	MW(WORD_STRONG := MesBlock1_Temp[1][  4], WORD_WEAK := MesBlock1_Temp[1][  3], VAR_OUT := MesDataExd.T1.MesI2);                       
	MW(WORD_STRONG := MesBlock1_Temp[1][  6], WORD_WEAK := MesBlock1_Temp[1][  5], VAR_OUT := MesDataExd.T1.MesI3);                       
	MW(WORD_STRONG := MesBlock1_Temp[1][  8], WORD_WEAK := MesBlock1_Temp[1][  7], VAR_OUT := MesDataExd.T1.MesU12);                      
	MW(WORD_STRONG := MesBlock1_Temp[1][ 10], WORD_WEAK := MesBlock1_Temp[1][  9], VAR_OUT := MesDataExd.T1.MesU23);                      
	MW(WORD_STRONG := MesBlock1_Temp[1][ 12], WORD_WEAK := MesBlock1_Temp[1][ 11], VAR_OUT := MesDataExd.T1.MesU31);                      
	MW(WORD_STRONG := MesBlock1_Temp[1][ 14], WORD_WEAK := MesBlock1_Temp[1][ 13], VAR_OUT := MesDataExd.T2.MesI1);                       
	MW(WORD_STRONG := MesBlock1_Temp[1][ 16], WORD_WEAK := MesBlock1_Temp[1][ 15], VAR_OUT := MesDataExd.T2.MesI2);                       
	MW(WORD_STRONG := MesBlock1_Temp[1][ 18], WORD_WEAK := MesBlock1_Temp[1][ 17], VAR_OUT := MesDataExd.T2.MesI3);                       
	MW(WORD_STRONG := MesBlock1_Temp[1][ 20], WORD_WEAK := MesBlock1_Temp[1][ 19], VAR_OUT := MesDataExd.T2.MesU12);                      
	MW(WORD_STRONG := MesBlock1_Temp[1][ 22], WORD_WEAK := MesBlock1_Temp[1][ 21], VAR_OUT := MesDataExd.T2.MesU23);                      
	MW(WORD_STRONG := MesBlock1_Temp[1][ 24], WORD_WEAK := MesBlock1_Temp[1][ 23], VAR_OUT := MesDataExd.T2.MesU31);                      
	MW(WORD_STRONG := MesBlock1_Temp[1][ 26], WORD_WEAK := MesBlock1_Temp[1][ 25], VAR_OUT := MesDataExd.T2.MesFreq );                             
	MW(WORD_STRONG := MesBlock1_Temp[1][ 28], WORD_WEAK := MesBlock1_Temp[1][ 27], VAR_OUT := MesDataExd.F11.MesEActProd);                                 
	MW(WORD_STRONG := MesBlock1_Temp[1][ 30], WORD_WEAK := MesBlock1_Temp[1][ 29], VAR_OUT := MesDataExd.F11.MesEActCons);                                 
	MW(WORD_STRONG := MesBlock1_Temp[1][ 32], WORD_WEAK := MesBlock1_Temp[1][ 31], VAR_OUT := MesDataExd.F11.MesEReactProd);               
	MW(WORD_STRONG := MesBlock1_Temp[1][ 34], WORD_WEAK := MesBlock1_Temp[1][ 33], VAR_OUT := MesDataExd.F11.MesEReactCons);                    
	MW(WORD_STRONG := MesBlock1_Temp[1][ 36], WORD_WEAK := MesBlock1_Temp[1][ 35], VAR_OUT := MesDataExd.F11.MesP);                       
	MW(WORD_STRONG := MesBlock1_Temp[1][ 38], WORD_WEAK := MesBlock1_Temp[1][ 37], VAR_OUT := MesDataExd.F11.MesQ);                       
	MW(WORD_STRONG := MesBlock1_Temp[1][ 40], WORD_WEAK := MesBlock1_Temp[1][ 39], VAR_OUT := MesDataExd.F11.MesU12);                     
	MW(WORD_STRONG := MesBlock1_Temp[1][ 42], WORD_WEAK := MesBlock1_Temp[1][ 41], VAR_OUT := MesDataExd.F11.MesU23);                     
	MW(WORD_STRONG := MesBlock1_Temp[1][ 44], WORD_WEAK := MesBlock1_Temp[1][ 43], VAR_OUT := MesDataExd.F11.MesU31);                     
	MW(WORD_STRONG := MesBlock1_Temp[1][ 46], WORD_WEAK := MesBlock1_Temp[1][ 45], VAR_OUT := MesDataExd.F11.MesV1);                      
	MW(WORD_STRONG := MesBlock1_Temp[1][ 48], WORD_WEAK := MesBlock1_Temp[1][ 47], VAR_OUT := MesDataExd.F11.MesV2);                      
	MW(WORD_STRONG := MesBlock1_Temp[1][ 50], WORD_WEAK := MesBlock1_Temp[1][ 49], VAR_OUT := MesDataExd.F11.MesV3);                      
	MW(WORD_STRONG := MesBlock1_Temp[1][ 52], WORD_WEAK := MesBlock1_Temp[1][ 51], VAR_OUT := MesDataExd.F11.MesI1);                      
	MW(WORD_STRONG := MesBlock1_Temp[1][ 54], WORD_WEAK := MesBlock1_Temp[1][ 53], VAR_OUT := MesDataExd.F11.MesI2);                      
	MW(WORD_STRONG := MesBlock1_Temp[1][ 56], WORD_WEAK := MesBlock1_Temp[1][ 55], VAR_OUT := MesDataExd.F11.MesI3);                   
	MW(WORD_STRONG := MesBlock1_Temp[1][ 58], WORD_WEAK := MesBlock1_Temp[1][ 57], VAR_OUT := MesDataExd.F11.MesFreq);                    
	MW(WORD_STRONG := MesBlock1_Temp[1][ 60], WORD_WEAK := MesBlock1_Temp[1][ 59], VAR_OUT := MesDataExd.F11.MesCosPhi);                
	MW(WORD_STRONG := MesBlock1_Temp[1][ 62], WORD_WEAK := MesBlock1_Temp[1][ 61], VAR_OUT := MesDataExd.F15.MesP);                 
	MW(WORD_STRONG := MesBlock1_Temp[1][ 64], WORD_WEAK := MesBlock1_Temp[1][ 63], VAR_OUT := MesDataExd.F15.MesQ);                 
	MW(WORD_STRONG := MesBlock1_Temp[1][ 66], WORD_WEAK := MesBlock1_Temp[1][ 65],  VAR_OUT :=MesDataExd.F15.MesI1);                     
	MW(WORD_STRONG := MesBlock1_Temp[1][ 68], WORD_WEAK := MesBlock1_Temp[1][ 67],  VAR_OUT :=MesDataExd.F15.MesI2);                  
	MW(WORD_STRONG := MesBlock1_Temp[1][ 70], WORD_WEAK := MesBlock1_Temp[1][ 69],  VAR_OUT :=MesDataExd.F15.MesI3);                  
	MW(WORD_STRONG := MesBlock1_Temp[1][ 72], WORD_WEAK := MesBlock1_Temp[1][ 71],  VAR_OUT :=MesDataExd.F15.MesU12);                 
	MW(WORD_STRONG := MesBlock1_Temp[1][ 74], WORD_WEAK := MesBlock1_Temp[1][ 73],  VAR_OUT :=MesDataExd.F15.MesU23);          
	MW(WORD_STRONG := MesBlock1_Temp[1][ 76], WORD_WEAK := MesBlock1_Temp[1][ 75],  VAR_OUT :=MesDataExd.F15.MesU31);    
	MW(WORD_STRONG := MesBlock1_Temp[1][ 78], WORD_WEAK := MesBlock1_Temp[1][ 77],  VAR_OUT :=MesDataExd.F15.MesV1);       
	MW(WORD_STRONG := MesBlock1_Temp[1][ 78], WORD_WEAK := MesBlock1_Temp[1][ 79],  VAR_OUT :=MesDataExd.F15.MesV2);       
	MW(WORD_STRONG := MesBlock1_Temp[1][ 80], WORD_WEAK := MesBlock1_Temp[1][ 81],  VAR_OUT :=MesDataExd.F15.MesV3);                
	MW(WORD_STRONG := MesBlock1_Temp[1][ 84], WORD_WEAK := MesBlock1_Temp[1][ 85],  VAR_OUT :=MesDataExd.F15.MesFreq);   

                    
	MW(WORD_STRONG := MesBlock1_Temp[2][ 22], WORD_WEAK := MesBlock1_Temp[2][21], VAR_OUT := MesDataExd.F21.MesEActProd);                      
	MW(WORD_STRONG := MesBlock1_Temp[2][ 24], WORD_WEAK := MesBlock1_Temp[2][23], VAR_OUT := MesDataExd.F21.MesEActCons);                      
	MW(WORD_STRONG := MesBlock1_Temp[2][ 26], WORD_WEAK := MesBlock1_Temp[2][25], VAR_OUT := MesDataExd.F21.MesEReactProd);                    
	MW(WORD_STRONG := MesBlock1_Temp[2][ 28], WORD_WEAK := MesBlock1_Temp[2][27], VAR_OUT := MesDataExd.F21.MesEReactCons);                    
	MW(WORD_STRONG := MesBlock1_Temp[2][ 30], WORD_WEAK := MesBlock1_Temp[2][29], VAR_OUT := MesDataExd.F21.MesP);                            
	MW(WORD_STRONG := MesBlock1_Temp[2][ 32], WORD_WEAK := MesBlock1_Temp[2][31], VAR_OUT := MesDataExd.F21.MesQ);                            
	MW(WORD_STRONG := MesBlock1_Temp[2][ 34], WORD_WEAK := MesBlock1_Temp[2][33], VAR_OUT := MesDataExd.F21.MesU12);                          
	MW(WORD_STRONG := MesBlock1_Temp[2][ 36], WORD_WEAK := MesBlock1_Temp[2][35], VAR_OUT := MesDataExd.F21.MesU23);                          
	MW(WORD_STRONG := MesBlock1_Temp[2][ 38], WORD_WEAK := MesBlock1_Temp[2][37], VAR_OUT := MesDataExd.F21.MesU31);                          
	MW(WORD_STRONG := MesBlock1_Temp[2][ 40], WORD_WEAK := MesBlock1_Temp[2][39], VAR_OUT := MesDataExd.F21.MesV1);                           
	MW(WORD_STRONG := MesBlock1_Temp[2][ 42], WORD_WEAK := MesBlock1_Temp[2][41], VAR_OUT := MesDataExd.F21.MesV2);                           
	MW(WORD_STRONG := MesBlock1_Temp[2][ 44], WORD_WEAK := MesBlock1_Temp[2][43], VAR_OUT := MesDataExd.F21.MesV3);                           
	MW(WORD_STRONG := MesBlock1_Temp[2][ 46], WORD_WEAK := MesBlock1_Temp[2][45], VAR_OUT := MesDataExd.F21.MesI1);                           
	MW(WORD_STRONG := MesBlock1_Temp[2][ 48], WORD_WEAK := MesBlock1_Temp[2][47], VAR_OUT := MesDataExd.F21.MesI2);                           
	MW(WORD_STRONG := MesBlock1_Temp[2][ 50], WORD_WEAK := MesBlock1_Temp[2][49], VAR_OUT := MesDataExd.F21.MesI3);                           
	MW(WORD_STRONG := MesBlock1_Temp[2][ 52], WORD_WEAK := MesBlock1_Temp[2][51], VAR_OUT := MesDataExd.F21.MesFreq);                         
	MW(WORD_STRONG := MesBlock1_Temp[2][ 54], WORD_WEAK := MesBlock1_Temp[2][53], VAR_OUT := MesDataExd.F21.MesCosPhi);                       
	MW(WORD_STRONG := MesBlock1_Temp[2][ 56], WORD_WEAK := MesBlock1_Temp[2][55], VAR_OUT := MesDataExd.F22.MesEActProd);                      
	MW(WORD_STRONG := MesBlock1_Temp[2][ 58], WORD_WEAK := MesBlock1_Temp[2][57], VAR_OUT := MesDataExd.F22.MesEActCons);                      
	MW(WORD_STRONG := MesBlock1_Temp[2][ 60], WORD_WEAK := MesBlock1_Temp[2][59], VAR_OUT := MesDataExd.F22.MesEReactProd);                    
	MW(WORD_STRONG := MesBlock1_Temp[2][ 62], WORD_WEAK := MesBlock1_Temp[2][61], VAR_OUT := MesDataExd.F22.MesEReactCons);                    
	MW(WORD_STRONG := MesBlock1_Temp[2][ 64], WORD_WEAK := MesBlock1_Temp[2][63], VAR_OUT := MesDataExd.F22.MesP);                            
	MW(WORD_STRONG := MesBlock1_Temp[2][ 66], WORD_WEAK := MesBlock1_Temp[2][65], VAR_OUT := MesDataExd.F22.MesQ);                            
	MW(WORD_STRONG := MesBlock1_Temp[2][ 68], WORD_WEAK := MesBlock1_Temp[2][67], VAR_OUT := MesDataExd.F22.MesU12);                          
	MW(WORD_STRONG := MesBlock1_Temp[2][ 70], WORD_WEAK := MesBlock1_Temp[2][69], VAR_OUT := MesDataExd.F22.MesU23);                          
	MW(WORD_STRONG := MesBlock1_Temp[2][ 72], WORD_WEAK := MesBlock1_Temp[2][71], VAR_OUT := MesDataExd.F22.MesU31);                          
	MW(WORD_STRONG := MesBlock1_Temp[2][ 74], WORD_WEAK := MesBlock1_Temp[2][73], VAR_OUT := MesDataExd.F22.MesV1);                           
	MW(WORD_STRONG := MesBlock1_Temp[2][ 76], WORD_WEAK := MesBlock1_Temp[2][75], VAR_OUT := MesDataExd.F22.MesV2);                           
	MW(WORD_STRONG := MesBlock1_Temp[2][ 78], WORD_WEAK := MesBlock1_Temp[2][77], VAR_OUT := MesDataExd.F22.MesV3);                           
	MW(WORD_STRONG := MesBlock1_Temp[2][ 80], WORD_WEAK := MesBlock1_Temp[2][79], VAR_OUT := MesDataExd.F22.MesI1);                           
	MW(WORD_STRONG := MesBlock1_Temp[2][ 82], WORD_WEAK := MesBlock1_Temp[2][81], VAR_OUT := MesDataExd.F22.MesI2);                           
	MW(WORD_STRONG := MesBlock1_Temp[2][ 84], WORD_WEAK := MesBlock1_Temp[2][83], VAR_OUT := MesDataExd.F22.MesI3);                           
	MW(WORD_STRONG := MesBlock1_Temp[2][ 86], WORD_WEAK := MesBlock1_Temp[2][85], VAR_OUT := MesDataExd.F22.MesFreq);                         
	MW(WORD_STRONG := MesBlock1_Temp[2][ 88], WORD_WEAK := MesBlock1_Temp[2][87], VAR_OUT := MesDataExd.F22.MesCosPhi); 

	MW(WORD_WEAK := MesBlock1_Temp[3][ 1], WORD_STRONG := MesBlock1_Temp[3][ 2], VAR_OUT := MesDataExd.T4.MesU12);
	MW(WORD_WEAK := MesBlock1_Temp[3][ 3], WORD_STRONG := MesBlock1_Temp[3][ 4], VAR_OUT := MesDataExd.T4.MesU23);
	MW(WORD_WEAK := MesBlock1_Temp[3][ 5], WORD_STRONG := MesBlock1_Temp[3][ 6], VAR_OUT := MesDataExd.T4.MesU31);
	                                                                              
	MW(WORD_WEAK := MesBlock1_Temp[4][ 1], WORD_STRONG := MesBlock1_Temp[4][ 2], VAR_OUT := MesDataExd.T5.MesU12);
	MW(WORD_WEAK := MesBlock1_Temp[4][ 3], WORD_STRONG := MesBlock1_Temp[4][ 4], VAR_OUT := MesDataExd.T5.MesU23);
	MW(WORD_WEAK := MesBlock1_Temp[4][ 5], WORD_STRONG := MesBlock1_Temp[4][ 6], VAR_OUT := MesDataExd.T5.MesU31);
	
MesDataExd.F11.MesU := (MesDataExd.F11.MesU12 + MesDataExd.F11.MesU23 + MesDataExd.F11.MesU31)/3 ;
MesDataExd.F11.MesI := (MesDataExd.F11.MesI1 + MesDataExd.F11.MesI2 + MesDataExd.F11.MesI3)/3 ;
MesDataExd.F11.MesV := (MesDataExd.F11.MesV1 + MesDataExd.F11.MesV2 + MesDataExd.F11.MesV3)/3 ;

MesDataExd.F15.MesU := (MesDataExd.F15.MesU12 + MesDataExd.F15.MesU23 + MesDataExd.F15.MesU31)/3 ;
MesDataExd.F15.MesI := (MesDataExd.F15.MesI1 + 	MesDataExd.F15.MesI2 + 	MesDataExd.F15.MesI3)/3 ;
MesDataExd.F15.MesV := (MesDataExd.F15.MesV1 + 	MesDataExd.F15.MesV2 + 	MesDataExd.F15.MesV3)/3 ;

MesDataExd.F21.MesU := (MesDataExd.F21.MesU12 + MesDataExd.F21.MesU23 + MesDataExd.F21.MesU31)/3 ;
MesDataExd.F21.MesI := (MesDataExd.F21.MesI1 + 	MesDataExd.F21.MesI2 + 	MesDataExd.F21.MesI3)/3 ;
MesDataExd.F21.MesV := (MesDataExd.F21.MesV1 + 	MesDataExd.F21.MesV2 + 	MesDataExd.F21.MesV3)/3 ;

MesDataExd.F22.MesU := (MesDataExd.F22.MesU12 + MesDataExd.F22.MesU23 + MesDataExd.F22.MesU31)/3 ;
MesDataExd.F22.MesI := (MesDataExd.F22.MesI1 + 	MesDataExd.F22.MesI2 + 	MesDataExd.F22.MesI3)/3 ;
MesDataExd.F22.MesV := (MesDataExd.F22.MesV1 + 	MesDataExd.F22.MesV2 + 	MesDataExd.F22.MesV3)/3 ;

MesDataExd.T1.MesU := (MesDataExd.T1.MesU12 + 	MesDataExd.T1.MesU23 + 	MesDataExd.T1.MesU31)/3 ;
MesDataExd.T1.MesI := (MesDataExd.T1.MesI1 + 	MesDataExd.T1.MesI2 + 	MesDataExd.T1.MesI3)/3 ;
MesDataExd.T1.MesV := (MesDataExd.T1.MesV1 + 	MesDataExd.T1.MesV2 + 	MesDataExd.T1.MesV3)/3 ;

MesDataExd.T2.MesU := (MesDataExd.T2.MesU12 + 	MesDataExd.T2.MesU23 + 	MesDataExd.T2.MesU31)/3 ;
MesDataExd.T2.MesI := (MesDataExd.T2.MesI1 + 	MesDataExd.T2.MesI2 + 	MesDataExd.T2.MesI3)/3 ;
MesDataExd.T2.MesV := (MesDataExd.T2.MesV1 + 	MesDataExd.T2.MesV2 + 	MesDataExd.T2.MesV3)/3 ;

MesDataExd.T4.MesU := (MesDataExd.T4.MesU12 + 	MesDataExd.T4.MesU23 + 	MesDataExd.T4.MesU31)/3 ;
MesDataExd.T5.MesU := (MesDataExd.T5.MesU12 + 	MesDataExd.T5.MesU23 + 	MesDataExd.T5.MesU31)/3 ;
END_METHOD

END_FUNCTION_BLOCK

// ---- 01_Equipement_Library/Operation Meter/FB_PM_520x230.TcPOU
FUNCTION_BLOCK FB_PM_520x230 EXTENDS FB_PM_Base
//////////////////
// Measurement Solution based on Digiware, but access through PMS Socomec
//////////////////
VAR CONSTANT
	// Characteristics of the object (Same for all instances)
			
END_VAR

VAR_INPUT PERSISTENT
	// Parameters of the Object (instance specific) 
	{attribute 'OPC.UA.DA' := '1'} 
	ParamUnitID					: BYTE := 1 ;									// (NA)unit ID
	ParamInInterfaceSub			: BOOL := TRUE; 								// Serial interface RS422/RS485 TYPE (0:EL6021,1:SUB9)			
END_VAR

VAR_OUTPUT
	//Child objects
	
END_VAR


VAR_INPUT 
			MesDataExd				: PM_Standard;								// (NA) Structure of the PM3250
END_VAR

VAR
	//M_ALARMMANAGEMENT VARIABLES//
	                                                    								
                                                        								

	//M_READ VARIABLES//
		ModbusRTU					: FB_ModbusRTU;								// (NA) FB for Modbus Reading


		ObjectCom					: INT;										// (NA) Sequence index
									
		Busy						: BOOL;
		StepRead					: UINT;										// (NA) Step for reading 2 blocks of registers
		AX_TrigRead					: ARRAY[1..1] OF R_trig;
		MbStruct					: ARRAY[1..1] OF Struct_InputRTU;	
		MesBlock					: ARRAY[1..1] OF ARRAY[1..120] OF WORD;	
		AX_Addr						: ARRAY[1..1] OF UINT 	:= [19000];
		AX_Qty						: ARRAY[1..1] OF UINT	:= [86];
		AX_UnitId					: ARRAY[1..1] OF BYTE	:= [1];
		AX_Function					: ARRAY[1..1] OF UINT	:= [4];	
		AX_Priority					: ARRAY[1..1] OF UINT	:= [1];
		KK							: INT;
		ComError 					: BOOL;
	//M_INIT VARIABLES //
		OutFBCompleteted			: BOOL;
	// M_EXECUTE VARIABLES //
		
                              

 
END_VAR

METHOD M_AlarmManagement
//////////////////
// Digiware measurement tool alarm and warning management
/////////////////

VAR 
	// Method local variables (reinitialized at each cycle) 
	FB_AlarmCodeManager			: FB_AlarmCodeManager ; 
	
	KK							: BYTE ;		// For loop
	
	CMWarning					: BOOL;			// At least one Digiware device in Alarm
	CMAlarm						: BOOL;			// At least one Digiware device in Alarm
	
END_VAR
//ComError 	:= MbStruct[1].OutError^;
	
TON_ComAlarm(IN:= ComError , PT:= ParamTempoComAlarm, Q=>MesDataExd.MesData.MesAlarmCom) ;	
TON_ComWarning(IN:= ComError  , PT:= ParamTempoComAlarm, Q=>MesWarningCom) ;	

//					General com alarm : All the read FB fucked up


// ALARM CODE //
	FB_AlarmCodeManager(
		bAlarm1			:= MesDataExd.MesData.MesAlarmCom  , 					// Communication Alarm #COM
		bAlarm2			:=FALSE, 		// 
		bAlarm3			:=FALSE, 		// 
		bAlarm4			:=FALSE, 		// 
		bAlarm5			:=FALSE, //
		bAlarm6			:=FALSE, //
		bAlarm7			:=FALSE, //
		bAlarm8			:=FALSE, //
		bAlarm9			:=FALSE, //
		bAlarm10		:=FALSE, //
		bAlarm11		:=FALSE, //
		bAlarm12		:=FALSE, //
		bAlarm13		:=FALSE, //
		bAlarm14		:=FALSE, //
		bAlarm15		:= FALSE , 			// 			 
		wAlarmCode		=>MesDataExd.MesData.MesAlarmCode);

// WARNING CODE //
	FB_AlarmCodeManager(		
		bAlarm1			:=MesWarningCom	,				 // Communication Warning #COM
		bAlarm2			:=FALSE, 		// 
		bAlarm3			:=FALSE, 		// 
		bAlarm4			:=FALSE, 		// 
		bAlarm5			:=FALSE, //
		bAlarm6			:=FALSE, //
		bAlarm7			:=FALSE, //
		bAlarm8			:=FALSE, //
		bAlarm9			:=FALSE, //
		bAlarm10		:=FALSE, //
		bAlarm11		:=FALSE, //
		bAlarm12		:=FALSE, //
		bAlarm13		:=FALSE, //
		bAlarm14		:=FALSE, //
		bAlarm15		:=FALSE, //
		wAlarmCode		=>MesDataExd.MesData.MesWarningCode);		

// EVENT CODE //
END_METHOD

METHOD M_CP
//////////////////
//  Emulator
/////////////////

VAR 
	// Method local variables (reinitialized at each cycle) 
	
END_VAR


SUPER^.M_CP() ; 




Trig_Cmd_Read(CLK:=IN_CmdToggleRead);
Trig_Cmd_Write(CLK:=IN_CmdToggleWrite);
	
IF Trig_Cmd_Read.Q THEN
	IN_CmdToggleRead := FALSE;
	MesDataExd.MesData.MesCP_Read := NOT MesDataExd.MesData.MesCP_Read;
END_IF


IF Trig_Cmd_Write.Q THEN
	IN_CmdToggleWrite := FALSE;
	MesDataExd.MesData.MesCP_Write := NOT MesDataExd.MesData.MesCP_Write;
END_IF
END_METHOD

METHOD M_Evaluate : BOOL
VAR_INPUT
END_VAR
END_METHOD

METHOD M_Execute
//////////////////
//  Method Calls 
/////////////////
VAR 
	// Method local variables (reinitialized at each cycle) 
	// EMULATOR
		Psoltot		: REAL;		// Total Solar Power . 
		KK			: BYTE;		// For Loop
	
END_VAR
// READING AND WRITING CLOCK //
	TP1(IN:=NOT TP1.Q , PT:= ParamClockReadTime);
	ClockRead 		:= TP1.Q;

// PERMANENT CONDITIONS //
	MesCP_Read 					:= TRUE  ; 
	
// METHODS CALLS //
	IF bInit THEN
		M_Init() ; 
		bInit					:= FALSE ; 
		
	END_IF

	M_Read() ; 
	
// EMULATOR COM READ  /////////////
	
	
	////////////////////
	M_AlarmManagement();
END_METHOD

METHOD M_Init
VAR 

END_VAR
//Modbus RTU Relay
FOR KK := 1 TO 1 DO 
	MbStruct[KK].InBuffer 		:= ADR(MesBlock[KK]);
	MbStruct[KK].InFunction 	:= AX_Function[KK];
	MbStruct[KK].InQuantity 	:= AX_Qty[KK];
	MbStruct[KK].InStartAddr 	:= AX_Addr[KK];
	MbStruct[KK].InUnitID 		:= AX_UnitId[KK];
	
END_FOR
END_METHOD

METHOD M_Read
//////////////////
//  Read Modbus Variable for PCS . 
/////////////////
VAR 
	// Method local variables (reinitialized at each cycle) 
	MW 					: FB_MergeWordsToFloat; 
	KK					: BYTE;  						// FOR Loop 

	
END_VAR
// CP-Read / Write 

MesDataExd.MesData.MesCP_Read := MesDataExd.MesData.MesCP_Read ; 
 

IF MesDataExd.MesData.MesCP_Read  THEN	

	ModbusRTU();
	
	
	FOR KK := 1 TO 1 DO
		AX_TrigRead[KK](CLK  :=ClockRead) ; // CalLocalTimeStruct.wSecond MOD 5 = 0);
		IF AX_TrigRead[KK].Q THEN
			ModbusRTU.M_AddAction_FIFO(InStruct := MbStruct[KK], InPriority := AX_Priority[KK]);
		END_IF
		MbStruct[KK].OutError			:= ADR(ComError);
	END_FOR  
							
	// PROPERTIES UPDATE // 
		// Block 1
	//MW( WORD_STRONG:= MesBlock_Temp[1][1], 	WORD_WEAK := MesBlock_Temp[1][2],	SIGNED:=TRUE, FIX:=0 , SIZE:=2, VAR_OUT := MesDataExd.MesData.MesI2);
		
	MW( WORD_STRONG:= MesBlock[1][1], 	WORD_WEAK := MesBlock[1][2], 	VAR_OUT:= MesDataExd.MesData.MesV1);
	MW( WORD_STRONG:= MesBlock[1][3], 	WORD_WEAK := MesBlock[1][4], 	VAR_OUT:= MesDataExd.MesData.MesV2);
	MW( WORD_STRONG:= MesBlock[1][5], 	WORD_WEAK := MesBlock[1][6], 	VAR_OUT:= MesDataExd.MesData.MesV3);
	MW( WORD_STRONG:= MesBlock[1][7], 	WORD_WEAK := MesBlock[1][8], 	VAR_OUT:= MesDataExd.MesData.MesU12);
	MW( WORD_STRONG:= MesBlock[1][9], 	WORD_WEAK := MesBlock[1][10], VAR_OUT:= MesDataExd.MesData.MesU23);
																					
	MW( WORD_STRONG:= MesBlock[1][11], 	WORD_WEAK := MesBlock[1][12], VAR_OUT:= MesDataExd.MesData.MesU31);
	MW( WORD_STRONG:= MesBlock[1][13], 	WORD_WEAK := MesBlock[1][14], VAR_OUT:= MesDataExd.MesData.MesI1);
	MW( WORD_STRONG:= MesBlock[1][15], 	WORD_WEAK := MesBlock[1][16], VAR_OUT:= MesDataExd.MesData.MesI2);
	MW( WORD_STRONG:= MesBlock[1][17], 	WORD_WEAK := MesBlock[1][18], VAR_OUT:= MesDataExd.MesData.MesI3);
	MW( WORD_STRONG:= MesBlock[1][19], 	WORD_WEAK := MesBlock[1][20], VAR_OUT:= MesDataExd.MesData.MesIN);
	MW( WORD_STRONG:= MesBlock[1][21], 	WORD_WEAK := MesBlock[1][22], VAR_OUT:= MesDataExd.MesData.MesP1);
	MW( WORD_STRONG:= MesBlock[1][23], 	WORD_WEAK := MesBlock[1][24], VAR_OUT:= MesDataExd.MesData.MesP2);
	MW( WORD_STRONG:= MesBlock[1][25], 	WORD_WEAK := MesBlock[1][26], VAR_OUT:= MesDataExd.MesData.MesP3);
																					
	MW( WORD_STRONG:= MesBlock[1][27], 	WORD_WEAK := MesBlock[1][28], VAR_OUT:= MesDataExd.MesData.MesP);
	MW( WORD_STRONG:= MesBlock[1][35], 	WORD_WEAK := MesBlock[1][36], VAR_OUT:= MesDataExd.MesData.MesS);
	MW( WORD_STRONG:= MesBlock[1][43], 	WORD_WEAK := MesBlock[1][44], VAR_OUT:= MesDataExd.MesData.MesQ);
	
	//MW( WORD_STRONG_F:= MesBlock[1][7], 	WORD_WEAK_F := MesBlock[1][8], NUMBER_F= MesDataExd.MesData.MesP);
	//MW( WORD_STRONG_F:= MesBlock[1][9], 	WORD_WEAK_F := MesBlock[1][10], NUMBER_F= MesDataExd.MesData.MesQ1);
	//MW( WORD_STRONG_F:= MesBlock[1][11], 	WORD_WEAK_F := MesBlock[1][12], NUMBER_F= MesDataExd.MesData.MesQ2);
	//MW( WORD_STRONG_F:= MesBlock[1][13], 	WORD_WEAK_F := MesBlock[1][14], NUMBER_F= MesDataExd.MesData.MesQ3);
	//MW( WORD_STRONG_F:= MesBlock[1][15], 	WORD_WEAK_F := MesBlock[1][16], NUMBER_F= MesDataExd.MesData.MesQ);
	//MW( WORD_STRONG_F:= MesBlock[1][23], 	WORD_WEAK_F := MesBlock[1][24], NUMBER_F= MesDataExd.MesData.MesS);
	
	//MW( WORD_STRONG_F:= MesBlock_Temp[4][1], 	WORD_WEAK_F := MesBlock_Temp[4][2], NUMBER_F= MesDataExd.MesData.MesTanPhi);
	//MW( WORD_STRONG_F:= MesBlock_Temp[4][3], 	WORD_WEAK_F := MesBlock_Temp[4][4], NUMBER_F= MesDataExd.MesData.MesFreq);
	//
	//MW( WORD_STRONG_F:= MesBlock_Temp[3][1], 	WORD_WEAK_F := MesBlock_Temp[3][2], NUMBER_F= MesDataExd.MesData.MesEActProd);
	//MW( WORD_STRONG_F:= MesBlock_Temp[3][3], 	WORD_WEAK_F := MesBlock_Temp[3][4], NUMBER_F= MesDataExd.MesData.MesEActCons);
	//MW( WORD_STRONG_F:= MesBlock_Temp[3][5], 	WORD_WEAK_F := MesBlock_Temp[3][6], NUMBER_F= MesDataExd.MesData.MesEReactProd);
	//MW( WORD_STRONG_F:= MesBlock_Temp[3][7], 	WORD_WEAK_F := MesBlock_Temp[3][8], NUMBER_F= MesDataExd.MesData.MesEReactCons);
	//MW( WORD_STRONG:= MesBlock_Temp[4][3], 	WORD_WEAK := MesBlock_Temp[4][4],	SIGNED:=TRUE, FIX:=0 , SIZE:=2, VAR_OUT := MesDataExd.MesData.MesFreq);
	//MW( WORD_STRONG:= MesBlock_Temp[5][1], 	WORD_WEAK := MesBlock_Temp[5][2],	SIGNED:=TRUE, FIX:=0 , SIZE:=2, VAR_OUT := MesDataExd.MesData.MesEActProd);
	//MW( WORD_STRONG:= MesBlock_Temp[5][3], 	WORD_WEAK := MesBlock_Temp[5][4],	SIGNED:=TRUE, FIX:=0 , SIZE:=2, VAR_OUT := MesDataExd.MesData.MesEActCons);
	//MW( WORD_STRONG:= MesBlock_Temp[5][5], 	WORD_WEAK := MesBlock_Temp[5][6],	SIGNED:=TRUE, FIX:=0 , SIZE:=2, VAR_OUT := MesDataExd.MesData.MesEReactProd);
	//MW( WORD_STRONG:= MesBlock_Temp[5][7], 	WORD_WEAK := MesBlock_Temp[5][8],	SIGNED:=TRUE, FIX:=0 , SIZE:=2, VAR_OUT := MesDataExd.MesData.MesEReactCons);
	MesDataExd.Mesdata.MesP	:= MesDataExd.MesData.MesP / 1000.0;
	MesDataExd.MesData.MesS	:= MesDataExd.MesData.MesS	/ 1000.0;
	MesDataExd.MesData.MesP 	:= -1 * MesDataExd.MesData.MesP;
	MesDataExd.MesData.MesP1 	:= -1 * MesDataExd.MesData.MesP1/ 1000.0;
	MesDataExd.MesData.MesP2 	:= -1 * MesDataExd.MesData.MesP2/ 1000.0;
	MesDataExd.MesData.MesP3 	:= -1 * MesDataExd.MesData.MesP3/ 1000.0;
	
	MesDataExd.MesData.MesQ 	:= -1 * MesDataExd.MesData.MesQ;
	
	MesDataExd.MesData.MesQ 	:= MesDataExd.MesData.MesQ/1000.0;
	
	IF MesDataExd.MesData.MesP <> 0 THEN
		MesDataExd.MesData.MesTanPhi := MesDataExd.MesData.MesQ /  MesDataExd.MesData.MesP;
	
	ELSE
		MesDataExd.MesData.MesTanPhi := 0;
	END_IF
	


END_IF
END_METHOD

END_FUNCTION_BLOCK

// ---- 01_Equipement_Library/Operation Meter/FB_PM_A40.TcPOU
FUNCTION_BLOCK FB_PM_A40 EXTENDS FB_PM_Base
//////////////////
// Measurement Solution based on Digiware, but access through PMS Socomec
//////////////////

VAR_INPUT PERSISTENT
	// Parameters of the Object (instance specific)
	{attribute 'OPC.UA.DA' := '1'}  
	ParamUnitID					: BYTE := 22; 										// (NA) All unit ID For the Device (I35 + 1 U20)                                                                    			
	{attribute 'OPC.UA.DA' := '1'}                                                                             			
	ParamIPAddress			   	: STRING := '192.168.20.15'; 						// (NA) IP Adress of D50 .
	{attribute 'OPC.UA.DA' := '1'} 
	ParamTCPPort				: UINT := 502;										// Modbus TCP Port


END_VAR

VAR_OUTPUT
	//Child objects
	
END_VAR

VAR_INPUT 
			MesDataExd				: PM_Standard;								// (NA) Structure of the PM3250
END_VAR

VAR
	//M_ALARMMANAGEMENT VARIABLES//
		
	//M_READ VARIABLES//
		FB_ModbusRead_I1			: ARRAY[1..2] OF  FB_ModbusRead ; 				// (NA) FB for Modbus Reading
	                                                                                    	
		MesBlock1_Temp 				: ARRAY[1..2] 	OF ARRAY[0..124] OF WORD;		//(NA) Temporary Block with multiple modbus reading (U30 + I35)
		MesModbusReadAlarm 		  	: ARRAY[1..2] OF BOOL ; 						// (NA) Modbus Read Alarm for communication 
		
		
		MesModbusAlarmCode			: ARRAY[1..2] OF UDINT;							// (NA) Modbus Read Alarm Code	
		
	//M_INIT VARIABLES //
		


 
END_VAR

METHOD M_AlarmManagement
//////////////////
// Digiware measurement tool alarm and warning management
/////////////////

VAR 
	// Method local variables (reinitialized at each cycle) 
	FB_AlarmCodeManager			: FB_AlarmCodeManager ; 
	
	KK							: BYTE ;		// For loop
	
	CMWarning					: BOOL;			// At least one Digiware device in Alarm
	CMAlarm						: BOOL;			// At least one Digiware device in Alarm
	
END_VAR
// COMMUNICATION // 

		CMWarning 		:= MesModbusReadAlarm[1] ;
		CMAlarm			:= MesModbusReadAlarm[1];
		
	// Warning
	MesWarningCom 		:= CMWarning ; 											// LOC with at least one Digiware module
	//Alarm
	TON_ComAlarm(IN:= CMAlarm, PT:= ParamTempoComAlarm, Q=>MesDataExd.MesData.MesAlarmCom) ;	 	// D50 LOC

// ALARM CODE //
	FB_AlarmCodeManager(
		bAlarm1			:=MesDataExd.MesData.MesAlarmCom , 					// Communication Alarm  #COM
		bAlarm2			:=FALSE, 									// 
		bAlarm3			:=FALSE, 									// 
		bAlarm4			:=FALSE, 									// 
		bAlarm5			:=FALSE, 									//
		bAlarm6			:=FALSE,                                    //
		bAlarm7			:=FALSE,                                    //
		bAlarm8			:=FALSE, 									//
		bAlarm9			:=FALSE,                                    //
		bAlarm10		:=FALSE,                                    //
		bAlarm11		:=FALSE, 									//
		bAlarm12		:=FALSE,                                    //
		bAlarm13		:=FALSE,                                    //
		bAlarm14		:=FALSE, 									//
		bAlarm15		:= FALSE , 									// 						 
		wAlarmCode		=>MesDataExd.MesData.MesAlarmCode);

// WARNING CODE //
	FB_AlarmCodeManager(		
		bAlarm1			:= MesWarningCom,				// Communication warning  #COM
		bAlarm2			:=FALSE, 						// 
		bAlarm3			:=FALSE, 						// 
		bAlarm4			:=FALSE, 						// 
		bAlarm5			:=FALSE, 						//
		bAlarm6			:=FALSE,                        //
		bAlarm7			:=FALSE,                        //
		bAlarm8			:=FALSE,                        //
		bAlarm9			:=FALSE,                        //
		bAlarm10		:=FALSE,                        //
		bAlarm11		:=FALSE,                        //
		bAlarm12		:=FALSE,                        //
		bAlarm13		:=FALSE,                        //
		bAlarm14		:=FALSE,                        //
		bAlarm15		:=FALSE,                        //
		wAlarmCode		=>MesDataExd.MesData.MesWarningCode);
END_METHOD

METHOD M_CP
//////////////////
//  Emulator
/////////////////

VAR 
	// Method local variables (reinitialized at each cycle) 
	
END_VAR


SUPER^.M_CP() ; 




Trig_Cmd_Read(CLK:=IN_CmdToggleRead);
Trig_Cmd_Write(CLK:=IN_CmdToggleWrite);
	
IF Trig_Cmd_Read.Q THEN
	IN_CmdToggleRead := FALSE;
	MesDataExd.MesData.MesCP_Read := NOT MesDataExd.MesData.MesCP_Read;
END_IF


IF Trig_Cmd_Write.Q THEN
	IN_CmdToggleWrite := FALSE;
	MesDataExd.MesData.MesCP_Write := NOT MesDataExd.MesData.MesCP_Write;
END_IF
END_METHOD

METHOD M_Read
//////////////////
//  Read Modbus Variable for PCS . 
/////////////////
VAR 
	// Method local variables (reinitialized at each cycle) 
	MW 					: FB_MergeWordsToDint; 
	KK					: BYTE;  						// FOR Loop 

	Pinterm				: REAL;
	Pinterm1			: REAL;
	Pinterm2			: REAL;
	Pinterm3			: REAL;
	Iinterm1			: REAL;
	Iinterm2			: REAL;
	Iinterm3			: REAL;
	IInterm				: REAL;
	QInterm1			: REAL;
	QInterm2			: REAL;
	QInterm3			: REAL;
	QInterm				: REAL;
	SInterm				: REAL;
END_VAR
//INITIALIZING MODBUS REQUESTS //
	FOR KK:=1 TO 2 DO
		FB_ModbusRead_I1[KK](Reset:= CmdClearFault_G ,sIPAddr:=ParamIPAddress, tTimeout:= ParamTimeout, 	nTCPport := ParamTCPPort	);
	
	END_FOR 

// CP-Read / Write 


IF MesDataExd.MesData.MesCP_Read  THEN		
// MODBUS REQUEST//
	FB_ModbusRead_I1[1](
		nQuantity		:= 89, 
		nMBAddr			:= 16#4800, 
		nUnitID			:= ParamUnitID,
		cbLength		:= SIZEOF(MesBlock1_Temp[1]) , 
		pDestAddr		:= ADR(MesBlock1_Temp[1]) ,
		ClockRead		:=  MesDataExd.MesData.MesCP_Read AND ClockRead ,
		ModbusReadAlarm	=>	MesModbusReadAlarm[1]);
		
		
		
	FB_ModbusRead_I1[2](
		nQuantity		:= 54, 
		nMBAddr			:= 16#4D80, 
		nUnitID			:= ParamUnitID,
		cbLength		:= SIZEOF(MesBlock1_Temp[2]) , 
		pDestAddr		:= ADR(MesBlock1_Temp[2]) ,
		ClockRead		:=  MesDataExd.MesData.MesCP_Read AND ClockRead ,
		ModbusReadAlarm	=>	MesModbusReadAlarm[2]);		
		
		
// PROPERTIES UPDATE // 
	
	// Block2
	MW(WORD_STRONG:= MesBlock1_Temp[1][4], WORD_WEAK := MesBlock1_Temp[1][5],SIGNED:=FALSE, FIX:=2 , SIZE:=2, VAR_OUT := MesDataExd.MesData.MesV);	
	MW(WORD_STRONG:= MesBlock1_Temp[1][6], WORD_WEAK := MesBlock1_Temp[1][7],SIGNED:=FALSE, FIX:=2 , SIZE:=2, VAR_OUT := MesDataExd.MesData.MesU);	
	MW(WORD_STRONG:= MesBlock1_Temp[1][8], WORD_WEAK := MesBlock1_Temp[1][9],SIGNED:=FALSE, FIX:=3 , SIZE:=2, VAR_OUT := MesDataExd.MesData.MesI);	
	MW(WORD_STRONG:= MesBlock1_Temp[1][10], WORD_WEAK := MesBlock1_Temp[1][11],SIGNED:=FALSE, FIX:=3 , SIZE:=2, VAR_OUT := MesDataExd.MesData.MesFreq);	
	MW(WORD_STRONG:= MesBlock1_Temp[1][12], WORD_WEAK := MesBlock1_Temp[1][13],SIGNED:=FALSE, FIX:=2 , SIZE:=2, VAR_OUT := MesDataExd.MesData.MesV1);	
	MW(WORD_STRONG:= MesBlock1_Temp[1][14], WORD_WEAK := MesBlock1_Temp[1][15],SIGNED:=FALSE, FIX:=2 , SIZE:=2, VAR_OUT := MesDataExd.MesData.MesV2);	
	MW(WORD_STRONG:= MesBlock1_Temp[1][16], WORD_WEAK := MesBlock1_Temp[1][17],SIGNED:=FALSE, FIX:=2 , SIZE:=2, VAR_OUT := MesDataExd.MesData.MesV3);	
	MW(WORD_STRONG:= MesBlock1_Temp[1][20], WORD_WEAK := MesBlock1_Temp[1][21],SIGNED:=FALSE, FIX:=2 , SIZE:=2, VAR_OUT := MesDataExd.MesData.MesU12);	
	MW(WORD_STRONG:= MesBlock1_Temp[1][22], WORD_WEAK := MesBlock1_Temp[1][23],SIGNED:=FALSE, FIX:=2 , SIZE:=2, VAR_OUT := MesDataExd.MesData.MesU23);	
	MW(WORD_STRONG:= MesBlock1_Temp[1][24], WORD_WEAK := MesBlock1_Temp[1][25],SIGNED:=FALSE, FIX:=2 , SIZE:=2, VAR_OUT := MesDataExd.MesData.MesU31);	
	MW(WORD_STRONG:= MesBlock1_Temp[1][26], WORD_WEAK := MesBlock1_Temp[1][27],SIGNED:=FALSE, FIX:=3 , SIZE:=2, VAR_OUT := MesDataExd.MesData.MesI1);	
	MW(WORD_STRONG:= MesBlock1_Temp[1][28], WORD_WEAK := MesBlock1_Temp[1][29],SIGNED:=FALSE, FIX:=3 , SIZE:=2, VAR_OUT := MesDataExd.MesData.MesI2);	
	MW(WORD_STRONG:= MesBlock1_Temp[1][30], WORD_WEAK := MesBlock1_Temp[1][31],SIGNED:=FALSE, FIX:=3 , SIZE:=2, VAR_OUT := MesDataExd.MesData.MesI3);
	MW(WORD_STRONG:= MesBlock1_Temp[1][44], WORD_WEAK := MesBlock1_Temp[1][45],SIGNED:=TRUE, FIX:=3 , SIZE:=2, VAR_OUT := MesDataExd.MesData.MesP);	
	MW(WORD_STRONG:= MesBlock1_Temp[1][46], WORD_WEAK := MesBlock1_Temp[1][47],SIGNED:=TRUE, FIX:=3 , SIZE:=2, VAR_OUT := MesDataExd.MesData.MesQ);	
	MW(WORD_STRONG:= MesBlock1_Temp[1][52], WORD_WEAK := MesBlock1_Temp[1][53],SIGNED:=FALSE, FIX:=3 , SIZE:=2, VAR_OUT := MesDataExd.MesData.MesS);	
	MW(WORD_STRONG:= MesBlock1_Temp[1][54],SIGNED:=TRUE, FIX:=3 , SIZE:=1, VAR_OUT := MesDataExd.MesData.MesCosPhi);		
	MW(WORD_STRONG:= MesBlock1_Temp[1][56], WORD_WEAK := MesBlock1_Temp[1][57],SIGNED:=TRUE, FIX:=3 , SIZE:=2, VAR_OUT := MesDataExd.MesData.MesP1);	
	MW(WORD_STRONG:= MesBlock1_Temp[1][58], WORD_WEAK := MesBlock1_Temp[1][59],SIGNED:=TRUE, FIX:=3 , SIZE:=2, VAR_OUT := MesDataExd.MesData.MesP2);	
	MW(WORD_STRONG:= MesBlock1_Temp[1][60], WORD_WEAK := MesBlock1_Temp[1][61],SIGNED:=TRUE, FIX:=3 , SIZE:=2, VAR_OUT := MesDataExd.MesData.MesP3);	
	MW(WORD_STRONG:= MesBlock1_Temp[1][62], WORD_WEAK := MesBlock1_Temp[1][63],SIGNED:=TRUE, FIX:=3 , SIZE:=2, VAR_OUT := MesDataExd.MesData.MesQ1);	
	MW(WORD_STRONG:= MesBlock1_Temp[1][64], WORD_WEAK := MesBlock1_Temp[1][65],SIGNED:=TRUE, FIX:=3 , SIZE:=2, VAR_OUT := MesDataExd.MesData.MesQ2);	
	MW(WORD_STRONG:= MesBlock1_Temp[1][66], WORD_WEAK := MesBlock1_Temp[1][67],SIGNED:=TRUE, FIX:=3 , SIZE:=2, VAR_OUT := MesDataExd.MesData.MesQ3);		
	MW(WORD_STRONG:= MesBlock1_Temp[1][80], WORD_WEAK := MesBlock1_Temp[1][81],SIGNED:=FALSE, FIX:=3 , SIZE:=2, VAR_OUT := MesDataExd.MesData.MesS1);	
	MW(WORD_STRONG:= MesBlock1_Temp[1][82], WORD_WEAK := MesBlock1_Temp[1][83],SIGNED:=FALSE, FIX:=3 , SIZE:=2, VAR_OUT := MesDataExd.MesData.MesS2);	
	MW(WORD_STRONG:= MesBlock1_Temp[1][84], WORD_WEAK := MesBlock1_Temp[1][85],SIGNED:=FALSE, FIX:=3 , SIZE:=2, VAR_OUT := MesDataExd.MesData.MesS3);	
	MW(WORD_STRONG:= MesBlock1_Temp[1][86],SIGNED:=TRUE, FIX:=3 , SIZE:=1, VAR_OUT := MesDataExd.MesData.MesCosPhi1);	
	MW(WORD_STRONG:= MesBlock1_Temp[1][87],SIGNED:=TRUE, FIX:=3 , SIZE:=1, VAR_OUT := MesDataExd.MesData.MesCosPhi2);
	MW(WORD_STRONG:= MesBlock1_Temp[1][88],SIGNED:=TRUE, FIX:=3 , SIZE:=1, VAR_OUT := MesDataExd.MesData.MesCosPhi3);
	

	// energies 
	MW(WORD_STRONG:= MesBlock1_Temp[2][4], WORD_WEAK := MesBlock1_Temp[2][5],SIGNED:=FALSE, FIX:=4 , SIZE:=2, VAR_OUT := MesDataExd.MesData.MesEActCons);
	MW(WORD_STRONG:= MesBlock1_Temp[2][7], WORD_WEAK := MesBlock1_Temp[2][8],SIGNED:=FALSE, FIX:=4 , SIZE:=2, VAR_OUT := MesDataExd.MesData.MesEActProd);	
	MW(WORD_STRONG:= MesBlock1_Temp[2][10], WORD_WEAK := MesBlock1_Temp[2][11],SIGNED:=FALSE, FIX:=4 , SIZE:=2, VAR_OUT := MesDataExd.MesData.MesEReactCons);
	MW(WORD_STRONG:= MesBlock1_Temp[2][13], WORD_WEAK := MesBlock1_Temp[2][14],SIGNED:=FALSE, FIX:=4 , SIZE:=2, VAR_OUT := MesDataExd.MesData.MesEReactProd);
	

END_IF

// Evaluate 
	IF MesDataExd.MesData.MesP > 0.01 OR MesDataExd.MesData.MesP < -0.01 THEN
		MesDataExd.MesData.MesTanPhi := MesDataExd.MesData.MesQ /MesDataExd.MesData.MesP;
	ELSE
		MesDataExd.MesData.MesTanPhi := 0;
	END_IF
END_METHOD

END_FUNCTION_BLOCK

// ---- 01_Equipement_Library/Operation Meter/FB_PM_Digiware.TcPOU
FUNCTION_BLOCK FB_PM_Digiware EXTENDS FB_PM_Base
//////////////////
// Measurement Solution based on Digiware, but access through PMS Socomec
//////////////////

VAR_INPUT PERSISTENT
	// Parameters of the Object (instance specific) 
	ParamUnitID					: BYTE	 	;						// (NA) U30 unit ID
	ParamIPAddress			   	: STRING 	;							// (NA) IP Adress of D50 .
	ParamTCPPort				: UINT 		;
	ParamInvertPower			: BOOL		;
END_VAR

VAR_OUTPUT
	//Child objects
	
END_VAR

VAR_INPUT 
			MesDataExd				: PM_DirisA40;								// (NA) Structure of the PM3250
END_VAR

VAR
	//M_ALARMMANAGEMENT VARIABLES//
		
	//M_READ VARIABLES//

		
		ModbusRead					: ARRAY[1..5] OF FB_ModbusRead ; 			// (NA) FB for Modbus Reading
		MesBlock1_Temp 				: ARRAY[1..5] OF ARRAY[1..120] OF WORD;		//(NA) Temporary Block with multiple modbus reading (U30 + I35)
		
		
	//M_CP VARIABLES //
		CmdWrite						: BOOL;
		Trig_Read						: R_TRIG;
		Trig_Write						: R_TRIG;

	// M_EXECUTE VARIABLES //

 
END_VAR

METHOD M_AlarmManagement
//////////////////
// Digiware measurement tool alarm and warning management
/////////////////

VAR 
	// Method local variables (reinitialized at each cycle) 
	FB_AlarmCodeManager			: FB_AlarmCodeManager ; 
	
	KK							: BYTE ;		// For loop
	
	
END_VAR
IF MesDataExd.MesData.MesCP_Read THEN
// COMMUNICATION // 
	TON_ComWarning(PT := ParamTempoComAlarm, IN := ModbusRead[1].ModbusReadAlarm OR ModbusRead[2].ModbusReadAlarm OR ModbusRead[3].ModbusReadAlarm) ; 											// LOC with at least one Digiware module
	TON_ComAlarm(PT := ParamTempoComAlarm, IN := ModbusRead[1].ModbusReadAlarm AND ModbusRead[2].ModbusReadAlarm AND ModbusRead[3].ModbusReadAlarm)	 ; 											// LOC with at least one Digiware module
ELSE
	TON_ComWarning(IN := FALSE);
	TON_ComAlarm(IN := FALSE);
END_IF

MesDataExd.MesComAlarm 	:= TON_ComAlarm.Q;
MesDataExd.MesComWarning 	:= TON_ComWarning.Q;

// ALARM CODE //
	FB_AlarmCodeManager(
		bAlarm1			:= MesDataExd.MesComAlarm, 			// Communication Error : All Modbus TCP Frame failed
		bAlarm2			:=FALSE, 							// 
		bAlarm3			:=FALSE, 							// 
		bAlarm4			:=FALSE, 							// 
		bAlarm5			:=FALSE, 							//  			
		bAlarm6			:=FALSE,  							// 
		bAlarm7			:=FALSE,  							// 
		bAlarm8			:=FALSE,  							// 
		bAlarm9			:=FALSE,  							// 
		bAlarm10		:=FALSE,  							// 
		bAlarm11		:=FALSE,  							// 
		bAlarm12		:=FALSE,  							// 
		bAlarm13		:=FALSE,  							// 
		bAlarm14		:=FALSE,  							// 
		bAlarm15		:=False , 							// 					 
		wAlarmCode		=> MesDataExd.MesData.MesAlarmCode);

// WARNING CODE //
	FB_AlarmCodeManager(		
		bAlarm1			:= MesDataExd.MesComWarning,				 	// Communication Warning : At least one Modbus TCP Frame failed
		bAlarm2			:=FALSE, 							// 
		bAlarm3			:=FALSE, 							// 
		bAlarm4			:=FALSE, 							// 
		bAlarm5			:=FALSE,  							// 
		bAlarm6			:=FALSE,  							// 
		bAlarm7			:=FALSE,  							// 
		bAlarm8			:=FALSE,  							// 
		bAlarm9			:=FALSE,  							// 
		bAlarm10		:=FALSE,  							// 
		bAlarm11		:=FALSE,  							// 
		bAlarm12		:=FALSE,  							// 
		bAlarm13		:=FALSE,  							// 
		bAlarm14		:=FALSE,  							// 
		bAlarm15		:=FALSE,  							// 
		wAlarmCode		=> MesDataExd.MesData.MesWarningCode);
END_METHOD

METHOD M_CP 
VAR_INPUT
END_VAR


SUPER^.M_CP() ; 




Trig_Cmd_Read(CLK:=IN_CmdToggleRead);
	
IF Trig_Cmd_Read.Q THEN
	IN_CmdToggleRead := FALSE;
	MesDataExd.MesData.MesCP_Read := NOT MesDataExd.MesData.MesCP_Read;
END_IF
END_METHOD

METHOD M_Init
VAR 

	KK: BYTE;
END_VAR
ParamTCPPort			:= 502;

MesDataExd.MesData.MesCP_Read := TRUE;
END_METHOD

METHOD M_Read
//////////////////
//  Read Modbus Variable for PCS . 
/////////////////
VAR 
	// Method local variables (reinitialized at each cycle) 
	MW 					: FB_MergeWordsToDint; 
	KK					: BYTE;  						// FOR Loop 

	AX_ADDR				: ARRAY[1.. 5] OF UINT := [50514, 	50780, 	51536];
	AX_QTY				: ARRAY[1.. 5] OF BYTE := [78,		46,		10];
	AX_UnitId			: ARRAY[1.. 5] OF BYTE := [1,		1,		1];
	
END_VAR
FOR KK := 1 TO 3 DO
	ModbusRead[KK]
	(
		sIPAddr := ParamIPAddress,
		pDestAddr := ADR(MesBlock1_Temp[KK]),
		tTimeout := ParamTimeout,
		nTcpPort := ParamTCPPort,
		nQuantity := AX_QTY[KK],
		cbLength := SIZEOF(MesBlock1_Temp[KK]),
		nUnitID := ParamUnitID,
		nMBAddr := AX_ADDR[KK],
		ClockRead := ClockRead AND MesDataExd.MesData.MesCP_Read
	);
END_FOR

IF MesDataExd.MesData.MesCP_Read THEN
// PROPERTIES UPDATE // 
	// Block 1
		MW(WORD_STRONG:= MesBlock1_Temp[1][ 1], WORD_WEAK := MesBlock1_Temp[1][ 2],	SIGNED:=FALSE, 	FIX:=2 , SIZE:=2, VAR_OUT:=MesDataExd.MesData.MesU12);
		MW(WORD_STRONG:= MesBlock1_Temp[1][ 3], WORD_WEAK := MesBlock1_Temp[1][ 4],	SIGNED:=FALSE, 	FIX:=2 , SIZE:=2, VAR_OUT:=MesDataExd.MesData.MesU23);
		MW(WORD_STRONG:= MesBlock1_Temp[1][ 5], WORD_WEAK := MesBlock1_Temp[1][ 6],	SIGNED:=FALSE, 	FIX:=2 , SIZE:=2, VAR_OUT:=MesDataExd.MesData.MesU31);
		MW(WORD_STRONG:= MesBlock1_Temp[1][ 7], WORD_WEAK := MesBlock1_Temp[1][ 8],	SIGNED:=FALSE, 	FIX:=2 , SIZE:=2, VAR_OUT:=MesDataExd.MesData.MesV1);
		MW(WORD_STRONG:= MesBlock1_Temp[1][ 9], WORD_WEAK := MesBlock1_Temp[1][10],	SIGNED:=FALSE, 	FIX:=2 , SIZE:=2, VAR_OUT:=MesDataExd.MesData.MesV2);
		MW(WORD_STRONG:= MesBlock1_Temp[1][11], WORD_WEAK := MesBlock1_Temp[1][12],	SIGNED:=FALSE, 	FIX:=2 , SIZE:=2, VAR_OUT:=MesDataExd.MesData.MesV3);
		MW(WORD_STRONG:= MesBlock1_Temp[1][13], WORD_WEAK := MesBlock1_Temp[1][14],	SIGNED:=FALSE, 	FIX:=2 , SIZE:=2, VAR_OUT:=MesDataExd.MesData.MesFreq);
		MW(WORD_STRONG:= MesBlock1_Temp[1][15], WORD_WEAK := MesBlock1_Temp[1][16],	SIGNED:=FALSE, 	FIX:=3 , SIZE:=2, VAR_OUT:=MesDataExd.Mesdata.MesI1);
		MW(WORD_STRONG:= MesBlock1_Temp[1][17], WORD_WEAK := MesBlock1_Temp[1][18],	SIGNED:=FALSE, 	FIX:=3 , SIZE:=2, VAR_OUT:=MesDataExd.Mesdata.MesI2);
		MW(WORD_STRONG:= MesBlock1_Temp[1][19], WORD_WEAK := MesBlock1_Temp[1][20],	SIGNED:=FALSE, 	FIX:=3 , SIZE:=2, VAR_OUT:=MesDataExd.Mesdata.MesI3);
		MW(WORD_STRONG:= MesBlock1_Temp[1][21], WORD_WEAK := MesBlock1_Temp[1][22],	SIGNED:=FALSE, 	FIX:=3 , SIZE:=2, VAR_OUT:=MesDataExd.Mesdata.mesIn);
		MW(WORD_STRONG:= MesBlock1_Temp[1][23], WORD_WEAK := MesBlock1_Temp[1][24],	SIGNED:=TRUE, 	FIX:=2 , SIZE:=2, VAR_OUT:=MesDataExd.Mesdata.mesP);
		MW(WORD_STRONG:= MesBlock1_Temp[1][25], WORD_WEAK := MesBlock1_Temp[1][26],	SIGNED:=TRUE, 	FIX:=2 , SIZE:=2, VAR_OUT:=MesDataExd.Mesdata.mesQ);
		MW(WORD_STRONG:= MesBlock1_Temp[1][27], WORD_WEAK := MesBlock1_Temp[1][28],	SIGNED:=FALSE, 	FIX:=2 , SIZE:=2, VAR_OUT:=MesDataExd.Mesdata.mesS);
		MW(WORD_STRONG:= MesBlock1_Temp[1][29], WORD_WEAK := MesBlock1_Temp[1][30],	SIGNED:=TRUE, 	FIX:=3 , SIZE:=2, VAR_OUT:=MesDataExd.Mesdata.MesCosPhi);
		MW(WORD_STRONG:= MesBlock1_Temp[1][31], WORD_WEAK := MesBlock1_Temp[1][32],	SIGNED:=TRUE, 	FIX:=2 , SIZE:=2, VAR_OUT:=MesDataExd.Mesdata.MesP1);
		MW(WORD_STRONG:= MesBlock1_Temp[1][33], WORD_WEAK := MesBlock1_Temp[1][34],	SIGNED:=TRUE, 	FIX:=2 , SIZE:=2, VAR_OUT:=MesDataExd.Mesdata.MesP2);
		MW(WORD_STRONG:= MesBlock1_Temp[1][35], WORD_WEAK := MesBlock1_Temp[1][36],	SIGNED:=TRUE, 	FIX:=2 , SIZE:=2, VAR_OUT:=MesDataExd.Mesdata.MesP3);
		MW(WORD_STRONG:= MesBlock1_Temp[1][37], WORD_WEAK := MesBlock1_Temp[1][38],	SIGNED:=TRUE, 	FIX:=2 , SIZE:=2, VAR_OUT:=MesDataExd.Mesdata.MesQ1);
		MW(WORD_STRONG:= MesBlock1_Temp[1][39], WORD_WEAK := MesBlock1_Temp[1][40],	SIGNED:=TRUE, 	FIX:=2 , SIZE:=2, VAR_OUT:=MesDataExd.Mesdata.MesQ2);
		MW(WORD_STRONG:= MesBlock1_Temp[1][41], WORD_WEAK := MesBlock1_Temp[1][42],	SIGNED:=TRUE, 	FIX:=2 , SIZE:=2, VAR_OUT:=MesDataExd.Mesdata.MesQ3);
		
	
	
	// Block2
		MW(WORD_STRONG:= MesBlock1_Temp[2][ 1], WORD_WEAK := MesBlock1_Temp[2][ 2], SIGNED:=FALSE, FIX:=0 , SIZE:=1, VAR_OUT:=MesDataExd.MesData.MesEActProd);
		MW(WORD_STRONG:= MesBlock1_Temp[2][ 3], WORD_WEAK := MesBlock1_Temp[2][ 4], SIGNED:=FALSE, FIX:=0 , SIZE:=1, VAR_OUT:=MesDataExd.MesData.MesEReactProd);
		MW(WORD_STRONG:= MesBlock1_Temp[2][ 7], WORD_WEAK := MesBlock1_Temp[2][ 8], SIGNED:=FALSE, FIX:=0 , SIZE:=1, VAR_OUT:=MesDataExd.MesData.MesEActCons);
		MW(WORD_STRONG:= MesBlock1_Temp[2][ 9], WORD_WEAK := MesBlock1_Temp[2][10], SIGNED:=FALSE, FIX:=0 , SIZE:=1, VAR_OUT:=MesDataExd.MesData.MesEReactCons);
	
	// Block3
		MW(WORD_STRONG:= MesBlock1_Temp[3][ 1], SIGNED:=FALSE, FIX:=2 , SIZE:=1, VAR_OUT:=MesDataExd.MesTHDU12);
		MW(WORD_STRONG:= MesBlock1_Temp[3][ 2], SIGNED:=FALSE, FIX:=2 , SIZE:=1, VAR_OUT:=MesDataExd.MesTHDU23);
		MW(WORD_STRONG:= MesBlock1_Temp[3][ 3], SIGNED:=FALSE, FIX:=2 , SIZE:=1, VAR_OUT:=MesDataExd.MesTHDU31);
		MW(WORD_STRONG:= MesBlock1_Temp[3][ 4], SIGNED:=FALSE, FIX:=2 , SIZE:=1, VAR_OUT:=MesDataExd.MesTHDV1);
		MW(WORD_STRONG:= MesBlock1_Temp[3][ 5], SIGNED:=FALSE, FIX:=2 , SIZE:=1, VAR_OUT:=MesDataExd.MesTHDV2);
		MW(WORD_STRONG:= MesBlock1_Temp[3][ 6], SIGNED:=FALSE, FIX:=2 , SIZE:=1, VAR_OUT:=MesDataExd.MesTHDV3);
		MW(WORD_STRONG:= MesBlock1_Temp[3][ 7], SIGNED:=FALSE, FIX:=2 , SIZE:=1, VAR_OUT:=MesDataExd.MesTHDI1);
		MW(WORD_STRONG:= MesBlock1_Temp[3][ 8], SIGNED:=FALSE, FIX:=2 , SIZE:=1, VAR_OUT:=MesDataExd.MesTHDI2);
		MW(WORD_STRONG:= MesBlock1_Temp[3][ 9], SIGNED:=FALSE, FIX:=2 , SIZE:=1, VAR_OUT:=MesDataExd.MesTHDI3);
		MW(WORD_STRONG:= MesBlock1_Temp[3][10], SIGNED:=FALSE, FIX:=2 , SIZE:=1, VAR_OUT:=MesDataExd.MesTHDIN);
		
	MesDataExd.MesData.MesI := (MesDataExd.Mesdata.MesI1 + MesDataExd.MesData.MesI2 + MesDataExd.MesData.mesI3)/3;
	MesDataExd.MesData.MesU := (MesDataExd.Mesdata.MesU12 + MesDataExd.MesData.MesU23 + MesDataExd.MesData.mesU31)/3;
	MesDataExd.MesData.MesV := (MesDataExd.MesData.MesV1 + MesDataExd.MesData.MesV2 + MesDataExd.mesdata.MesV3)/3;
	IF ParamInvertPower THEN
		MesDataExd.MesData.MesP 	:= - MesDataExd.MesData.MesP;
		MesDataExd.MesData.MesP1 	:= - MesDataExd.MesData.MesP1;
		MesDataExd.MesData.MesP2 	:= - MesDataExd.MesData.MesP2;
		MesDataExd.MesData.MesP3 	:= - MesDataExd.MesData.MesP3;
		MesDataExd.MesData.MesQ 	:= - MesDataExd.MesData.MesQ;
		MesDataExd.MesData.MesQ1 	:= - MesDataExd.MesData.MesQ1;
		MesDataExd.MesData.MesQ2 	:= - MesDataExd.MesData.MesQ2;
		MesDataExd.MesData.MesQ3 	:= - MesDataExd.MesData.MesQ3;
	END_IF
END_IF
END_METHOD

END_FUNCTION_BLOCK

// ---- 01_Equipement_Library/Operation Meter/FB_PM_ION7650.TcPOU
FUNCTION_BLOCK FB_PM_ION7650 EXTENDS FB_PM_Base
//////////////////
// Measurement Solution based on Digiware, but access through PMS Socomec
//////////////////
VAR CONSTANT
	// Characteristics of the object (Same for all instances)
			
END_VAR

VAR_INPUT PERSISTENT
	// Parameters of the Object (instance specific) 
	{attribute 'OPC.UA.DA' := '1'} 
	ParamUnitID					: BYTE 		:= 1 ;								(* (NA) Unit ID*)
//	ParamInInterfaceSub			: BOOL 		:= TRUE; 							// (NA) Serial interface RS422/RS485 TYPE (0:EL6021,1:SUB9)
	{attribute 'OPC.UA.DA' := '1'} 
	ParamIPAddress		   		: STRING 	:= '192.168.20.15'; 				(* (NA) IP Adress of ION7650 *)
	{attribute 'OPC.UA.DA' := '1'} 
	ParamTcpPort				: UINT 		:= 502;								(* (NA) TCP port			*)
	ParamPCountZero				: INT		:= 1;								(* (NA) Number of time the PM P measurement was reinitialized to zero *)

END_VAR

VAR_OUTPUT
	//Child objects
	
END_VAR

VAR_INPUT 
			MesDataExd				: PM_Standard;								// (NA) Structure of the PM3250
END_VAR

VAR                                                  								                                          								
	//M_READ VARIABLES//
		FB_ModbusRead				: FB_ModbusRTU ;						// (NA) FB for Modbus Reading
		InputStructRead 			: ARRAY[1..1] OF  Struct_InputRTU;
		
		AX_Quantity					: ARRAY[1..1] OF WORD;					// (NA) Quantity of blocks to read
		AX_Address					: ARRAY[1..1] OF WORD;					// (NA) Start address of the read
		MesBlock_Temp 				: ARRAY[1..1] OF ARRAY[1..125] OF WORD;	// (NA) Temporary Block with multiple modbus reading (U30 + I35)
		Busy						: BOOL;
		OutErrorMbRead				: ARRAY[1..1] OF BOOL;
		
		RTrigI						: R_TRIG;
	//M_INIT VARIABLES //
		OutFBCompleteted			: BOOL;
	// ION was reset to 0 
		IONCount_PossibleReset		: BOOL := TRUE; 						// (NA) The active power of the PM ION7650 is between 1000 and  10m 
		
		
		
END_VAR

METHOD M_AlarmManagement
//////////////////
// Digiware measurement tool alarm and warning management
/////////////////

VAR 
	// Method local variables (reinitialized at each cycle) 
	FB_AlarmCodeManager			: FB_AlarmCodeManager ; 
	
	KK							: BYTE ;		// For loop
	
	CMWarning					: BOOL;			// At least one Digiware device in Alarm
	CMAlarm						: BOOL;			// At least one Digiware device in Alarm
	
END_VAR
TON_ComAlarm(IN:= OutErrorMbRead[1], PT:= ParamTempoComAlarm, Q=>MesDataExd.MesData.MesAlarmCom) ;	
//					General com alarm : All the read FB fucked up

// ALARM CODE //
	FB_AlarmCodeManager( 
		bAlarm1			:=MesDataExd.MesData.MesAlarmCom, 					// Communication Error  #COM
		bAlarm2			:=FALSE, 									// 
		bAlarm3			:=FALSE, 									// 
		bAlarm4			:=FALSE, 									// 
		bAlarm5			:=FALSE, 									//
		bAlarm6			:=FALSE, 									//
		bAlarm7			:=FALSE, 									//
		bAlarm8			:=FALSE, 									//
		bAlarm9			:=FALSE, 									//
		bAlarm10		:=FALSE, 									//
		bAlarm11		:=FALSE, 									//
		bAlarm12		:=FALSE, 									//
		bAlarm13		:=FALSE, 									//
		bAlarm14		:=FALSE, 									//
		bAlarm15		:= FALSE , 									//						 
		wAlarmCode		=>MesDataExd.MesData.MesAlarmCode);

// WARNING CODE //
	FB_AlarmCodeManager(		
		bAlarm1			:=	MesWarningCom,				 			// Communication Warning #COM	
		bAlarm2			:=FALSE, 									// 
		bAlarm3			:=FALSE, 									// 
		bAlarm4			:=FALSE, 									// 
		bAlarm5			:=FALSE, 									//
		bAlarm6			:=FALSE, 									//
		bAlarm7			:=FALSE, 									//
		bAlarm8			:=FALSE, 									//
		bAlarm9			:=FALSE, 									//
		bAlarm10		:=FALSE, 									//
		bAlarm11		:=FALSE, 									//
		bAlarm12		:=FALSE, 									//
		bAlarm13		:=FALSE, 									//
		bAlarm14		:=FALSE, 									//
		bAlarm15		:=FALSE, 									//
		wAlarmCode		=>MesDataExd.MesData.MesWarningCode);
END_METHOD

METHOD M_CP 
VAR_INPUT
END_VAR


SUPER^.M_CP() ; 




Trig_Cmd_Read(CLK:=IN_CmdToggleRead);
	
IF Trig_Cmd_Read.Q THEN
	IN_CmdToggleRead := FALSE;
	MesDataExd.MesData.MesCP_Read := NOT MesDataExd.MesData.MesCP_Read;
END_IF
END_METHOD

METHOD M_Evaluate : BOOL
VAR_INPUT
END_VAR
END_METHOD

METHOD M_Init
VAR 

END_VAR
(*FB_ModbusRead(InTimeout:= ParamTimeout,
				 InUnitID:= DINT_TO_BYTE(ParamUnitID),
				 InQuantity:= 125,	
				 InInterfaceSub:= ParamInInterfaceSub,
				 InFunctionRead := FALSE);
*)
	
AX_Quantity[1] := 125;
AX_Address[1]  := 149;
END_METHOD

METHOD M_Read
//////////////////
//  Read Modbus Variable for ION7650. 
/////////////////
VAR 
	// Method local variables (reinitialized at each cycle) 
	MW 					: FB_MergeWordsToDint; 
	KK					: BYTE;  						// FOR Loop 

END_VAR
// CP-Read / Write 

 

IF MesDataExd.MesData.MesCP_Read  THEN	
// MODBUS REQUEST TCP-IP //
(*	 
	ModbusRead
	(
		pDestAddr := ADR(MesBlock1_Temp),
		sIPAddr := ParamIPAdress,
		tTimeout := ParamTimeout,
		nQuantity := 122,
		nMBAddr := 150,
		cbLength := SIZEOF(MesBlock1_Temp),
		nUnitID := ParamUnitID,
		ClockRead := ClockRead,
		ErrorId => ModbusAlarmsID,
		ModbusReadAlarm => ModbusAlarm
	);
	*)
// MODBUS REQUEST RTU //	
	FB_ModbusRead();

	RTrigI(CLK:= ClockRead );
//Metrology
	FOR KK:=1 TO 1 DO
		InputStructRead[KK].InBuffer := ADR(MesBlock_Temp[KK]);
		InputStructRead[KK].InFunction := 3;
		InputStructRead[KK].InQuantity := AX_Quantity[KK];
		InputStructRead[KK].InStartAddr := AX_Address[KK];
		InputStructRead[KK].InUnitID := ParamUnitID;
		
		InputStructRead[KK].OutBusy := ADR(Busy);
		InputStructRead[KK].OutError := ADR(OutErrorMbRead[KK]);
		//InputStructRead[KK].OutCompleted := ADR(bReadCompleted);
		
		IF RTrigI.Q THEN 
			FB_ModbusRead.M_AddAction_FIFO(InStruct:= InputStructRead[KK] , InPriority:=1 ) ; 
		END_IF
		
	END_FOR 
				
// PROPERTIES UPDATE // 
	// Block 1
	MW(WORD_STRONG:= MesBlock_Temp[1][  1], SIGNED:=FALSE, FIX:=1 , SIZE:=1, 	VAR_OUT	:= MesDataExd.MesData.MesI1);
	MW(WORD_STRONG:= MesBlock_Temp[1][  2], SIGNED:=FALSE, FIX:=1 , SIZE:=1, 	VAR_OUT	:= MesDataExd.MesData.MesI2);
	MW(WORD_STRONG:= MesBlock_Temp[1][  3], SIGNED:=FALSE, FIX:=1 , SIZE:=1, 	VAR_OUT	:= MesDataExd.MesData.MesI3);
	MW(WORD_STRONG:= MesBlock_Temp[1][  6], SIGNED:=FALSE, FIX:=1 , SIZE:=1, 	VAR_OUT	:= MesDataExd.MesData.MesI);
	MW(WORD_STRONG:= MesBlock_Temp[1][ 10], SIGNED:=FALSE, FIX:=1 , SIZE:=1, 	VAR_OUT	:= MesDataExd.MesData.MesFreq);
	MW(WORD_STRONG:= MesBlock_Temp[1][ 17], Word_WEAK:= MesBlock_Temp[1][ 18], 	SIGNED:=FALSE, FIX:=0 , SIZE:=2, VAR_OUT:= MesDataExd.MesData.MesV1);
	MW(WORD_STRONG:= MesBlock_Temp[1][ 19], Word_WEAK:= MesBlock_Temp[1][ 20], 	SIGNED:=FALSE, FIX:=0 , SIZE:=2, VAR_OUT:= MesDataExd.MesData.MesV2);
	MW(WORD_STRONG:= MesBlock_Temp[1][ 21], Word_WEAK:= MesBlock_Temp[1][ 22], 	SIGNED:=FALSE, FIX:=0 , SIZE:=2, VAR_OUT:= MesDataExd.MesData.MesV3);
	MW(WORD_STRONG:= MesBlock_Temp[1][ 23], Word_WEAK:= MesBlock_Temp[1][ 24], 	SIGNED:=FALSE, FIX:=0 , SIZE:=2, VAR_OUT:= MesDataExd.MesData.MesV);
	MW(WORD_STRONG:= MesBlock_Temp[1][ 29], Word_WEAK:= MesBlock_Temp[1][ 30], 	SIGNED:=FALSE, FIX:=0 , SIZE:=2, VAR_OUT:= MesDataExd.MesData.MesU12);
	MW(WORD_STRONG:= MesBlock_Temp[1][ 31], Word_WEAK:= MesBlock_Temp[1][ 32], 	SIGNED:=FALSE, FIX:=0 , SIZE:=2, VAR_OUT:= MesDataExd.MesData.MesU23);
	MW(WORD_STRONG:= MesBlock_Temp[1][ 33], Word_WEAK:= MesBlock_Temp[1][ 34], 	SIGNED:=FALSE, FIX:=0 , SIZE:=2, VAR_OUT:= MesDataExd.MesData.MesU31);
	MW(WORD_STRONG:= MesBlock_Temp[1][ 35], Word_WEAK:= MesBlock_Temp[1][ 36], 	SIGNED:=FALSE, FIX:=0 , SIZE:=2, VAR_OUT:= MesDataExd.MesData.MesU);	
	MW(WORD_STRONG:= MesBlock_Temp[1][ 49], Word_WEAK:= MesBlock_Temp[1][ 50], 	SIGNED:=TRUE , FIX:=0 , SIZE:=2, VAR_OUT:= MesDataExd.MesData.MesP1);
	MW(WORD_STRONG:= MesBlock_Temp[1][ 51], Word_WEAK:= MesBlock_Temp[1][ 52], 	SIGNED:=TRUE , FIX:=0 , SIZE:=2, VAR_OUT:= MesDataExd.MesData.MesP2);
	MW(WORD_STRONG:= MesBlock_Temp[1][ 53], Word_WEAK:= MesBlock_Temp[1][ 54], 	SIGNED:=TRUE , FIX:=0 , SIZE:=2, VAR_OUT:= MesDataExd.MesData.MesP3);
	MW(WORD_STRONG:= MesBlock_Temp[1][ 55], Word_WEAK:= MesBlock_Temp[1][ 56], 	SIGNED:=TRUE , FIX:=0 , SIZE:=2, VAR_OUT:= MesDataExd.MesData.MesP);	
	MW(WORD_STRONG:= MesBlock_Temp[1][ 59], Word_WEAK:= MesBlock_Temp[1][ 60], 	SIGNED:=TRUE , FIX:=0 , SIZE:=2, VAR_OUT:= MesDataExd.MesData.MesQ1);	
	MW(WORD_STRONG:= MesBlock_Temp[1][ 61], Word_WEAK:= MesBlock_Temp[1][ 62], 	SIGNED:=TRUE , FIX:=0 , SIZE:=2, VAR_OUT:= MesDataExd.MesData.MesQ2);	
	MW(WORD_STRONG:= MesBlock_Temp[1][ 63], Word_WEAK:= MesBlock_Temp[1][ 64], 	SIGNED:=TRUE , FIX:=0 , SIZE:=2, VAR_OUT:= MesDataExd.MesData.MesQ3);	
	MW(WORD_STRONG:= MesBlock_Temp[1][ 65], Word_WEAK:= MesBlock_Temp[1][ 66], 	SIGNED:=TRUE , FIX:=0 , SIZE:=2, VAR_OUT:= MesDataExd.MesData.MesQ);	
	MW(WORD_STRONG:= MesBlock_Temp[1][ 75], Word_WEAK:= MesBlock_Temp[1][ 76], 	SIGNED:=TRUE , FIX:=0 , SIZE:=2, VAR_OUT:= MesDataExd.MesData.MesS);	
	                                                                                                                       
	MW(WORD_STRONG:= MesBlock_Temp[1][ 81], Word_weak:= MesBlock_Temp[1][ 82], 	SIGNED:=TRUE , FIX:=0 , SIZE:=2, VAR_OUT:= MesDataExd.MesData.MesEActProd);
	MW(WORD_STRONG:= MesBlock_Temp[1][ 83], Word_weak:= MesBlock_Temp[1][ 84], 	SIGNED:=TRUE , FIX:=0 , SIZE:=2, VAR_OUT:= MesDataExd.MesData.MesEActCons);
	MW(WORD_STRONG:= MesBlock_Temp[1][ 85], Word_weak:= MesBlock_Temp[1][ 86], 	SIGNED:=TRUE , FIX:=0 , SIZE:=2, VAR_OUT:= MesDataExd.MesData.MesEReactProd);
	MW(WORD_STRONG:= MesBlock_Temp[1][ 87], Word_weak:= MesBlock_Temp[1][ 88], 	SIGNED:=TRUE , FIX:=0 , SIZE:=2, VAR_OUT:= MesDataExd.MesData.MesEReactCons);
	                                                                 
	MW(WORD_STRONG:= MesBlock_Temp[1][113], SIGNED:=FALSE , FIX:=4 , SIZE:=1,	VAR_OUT:= MesDataExd.MesData.MesCosPhi1);
	MW(WORD_STRONG:= MesBlock_Temp[1][114], SIGNED:=FALSE , FIX:=4 , SIZE:=1,	VAR_OUT:= MesDataExd.MesData.MesCosPhi2);
	MW(WORD_STRONG:= MesBlock_Temp[1][115], SIGNED:=FALSE , FIX:=4 , SIZE:=1,	VAR_OUT:= MesDataExd.MesData.MesCosPhi3);
	MW(WORD_STRONG:= MesBlock_Temp[1][116], SIGNED:=FALSE , FIX:=4 , SIZE:=1,	VAR_OUT:= MesDataExd.MesData.MesCosPhi);
	
	
// Add the previous produced energy before counter reset
	IF MesDataExd.MesData.MesEActProd > 0 AND MesDataExd.MesData.MesEActProd < 1000  AND IONCount_PossibleReset THEN  
		IONCount_PossibleReset := FALSE;
		ParamPCountZero := ParamPCountZero + 1;	
	ELSIF MesDataExd.MesData.MesEActProd > 1000 THEN
		IONCount_PossibleReset := TRUE;
	END_IF

MesDataExd.MesData.MesEActProd := MesDataExd.MesData.MesEActProd + 10000000*ParamPCountZero;	
		
	IF MesDataExd.MesData.MesP<0.01 AND MesDataExd.MesData.MesP>-0.01  THEN 
		MesDataExd.MesData.MesTanPhi := 0 ;  
	ELSE
		MesDataExd.MesData.MesTanPhi := MesDataExd.MesData.MesQ /MesDataExd.MesData.MesP ; 
	END_IF
	
END_IF
END_METHOD

END_FUNCTION_BLOCK

// ---- 01_Equipement_Library/Operation Meter/FB_PM_Janitza.TcPOU
FUNCTION_BLOCK FB_PM_Janitza EXTENDS FB_PM_Base
//////////////////
// Measurement Solution based on Janitza, but access through JemaPLC
//////////////////

VAR_INPUT PERSISTENT
	// Parameters of the Object (instance specific) 
	{attribute 'OPC.UA.DA' := '1'} 
	ParamIpAddress			   	: STRING 		:= '192.168.1.30'; 			(* (NA) IP Adress of D50 .*)
	{attribute 'OPC.UA.DA' := '1'} 
	ParamUnitID 				: BYTE  := 1; 			  					(* (NA)   Modbus Unit ID.	*)


END_VAR

VAR_OUTPUT
	//Child objects
	
END_VAR

VAR_INPUT 
				MesDataExd AT %Q*				: PM_Standard ;
END_VAR

VAR
	//M_ALARMMANAGEMENT VARIABLES//
	
	//M_READ VARIABLES//
		FB_ModbusRead_I1			: ARRAY[1..1] OF  FB_ModbusRead ; 		// (NA) FB for Modbus Reading
	
		MesBlock1_Temp 				: ARRAY[0..125] OF WORD;				//(NA) Temporary Block with multiple modbus reading (U30 + I35)
		
		MesModbusReadAlarm 		  	: ARRAY[1..1] OF BOOL ; 				// (NA) Modbus Read Alarm for communication 
		
		MesModbusAlarmCode			: UDINT;								// (NA) Modbus Read Alarm Code	
		
	//M_INIT VARIABLES //

	// M_EXECUTE VARIABLES //

	
END_VAR

METHOD M_AlarmManagement
//////////////////
// Digiware measurement tool alarm and warning management
/////////////////

VAR 
	// Method local variables (reinitialized at each cycle) 
	FB_AlarmCodeManager			: FB_AlarmCodeManager ; 
	
	KK							: BYTE ;		// For loop
	
	CMWarning					: BOOL;			// At least one Digiware device in Alarm
	CMAlarm						: BOOL;			// At least one Digiware device in Alarm
	
END_VAR
// COMMUNICATION // 
IF MesDataExd.MesData.MesCP_Read then
	CMWarning 			:= FALSE ;
	CMAlarm	 			:= TRUE ;
	
	FOR KK:=1 TO 1 DO
		CMWarning 		:= CMWarning OR MesModbusReadAlarm[KK] ;
		CMAlarm			:= CMAlarm AND MesModbusReadAlarm[KK] ; 
	END_FOR
END_IF
	
	// Warning
	MesWarningCom 		:= CMWarning ; 											// LOC with at least one Digiware module
	//Alarm
	TON_ComAlarm(IN:= CMAlarm , PT:= ParamTempoComAlarm, Q=>MesDataExd.MesData.MesAlarmCom) ;	 	// D50 LOC

// ALARM CODE //
	FB_AlarmCodeManager(
		bAlarm1			:= MesDataExd.MesData.MesAlarmCom  , 					// Communication Alarm  #COM
		bAlarm2			:=FALSE, 		                            // 
		bAlarm3			:=FALSE, 		                            // 
		bAlarm4			:=FALSE, 		                            // 
		bAlarm5			:=FALSE,                                    //
		bAlarm6			:=FALSE,                                    //
		bAlarm7			:=FALSE,                                    //
		bAlarm8			:=FALSE,                                    //
		bAlarm9			:=FALSE,                                    //
		bAlarm10		:=FALSE,                                    //
		bAlarm11		:=FALSE,                                    //
		bAlarm12		:=FALSE,                                    //
		bAlarm13		:=FALSE,                                    //
		bAlarm14		:=FALSE,                                    //
		bAlarm15		:= FALSE , 			 						// 						 	 
		wAlarmCode		=>MesDataExd.MesData.MesAlarmCode);

// WARNING CODE //
	FB_AlarmCodeManager(		
		bAlarm1			:= MesWarningCom	,				// Communication warning  #COM
		bAlarm2			:=FALSE, 		                 	// 
		bAlarm3			:=FALSE, 		                  	// 
		bAlarm4			:=FALSE, 		                 	// 
		bAlarm5			:=FALSE,                            //
		bAlarm6			:=FALSE,                            //
		bAlarm7			:=FALSE,                            //
		bAlarm8			:=FALSE,                            //
		bAlarm9			:=FALSE,                            //
		bAlarm10		:=FALSE,                            //
		bAlarm11		:=FALSE,                            //
		bAlarm12		:=FALSE,                            //
		bAlarm13		:=FALSE,                            //
		bAlarm14		:=FALSE,                            //
		bAlarm15		:=FALSE,                            //
		wAlarmCode		=>MesDataExd.MesData.MesWarningCode);
END_METHOD

METHOD M_CP
//////////////////
//  Emulator
/////////////////

VAR 
	// Method local variables (reinitialized at each cycle) 
	
END_VAR


SUPER^.M_CP() ; 




Trig_Cmd_Read(CLK:=IN_CmdToggleRead);
	
IF Trig_Cmd_Read.Q THEN
	IN_CmdToggleRead := FALSE;
	MesDataExd.MesData.MesCP_Read := NOT MesDataExd.MesData.MesCP_Read;
END_IF
END_METHOD

METHOD M_Read
//////////////////
//  Read Modbus Variable for PCS . 
/////////////////
VAR 
	// Method local variables (reinitialized at each cycle) 
	MW 			: FB_MergeWordsToFloat ;
	
	MesPW	 : REAL ; 
	MesP1W   : REAL ; 
	MesP2W   : REAL ; 
	MesP3W   : REAL ; 
	MesQ1W   : REAL ; 
	MesQ2W   : REAL ; 
	MesQ3W   : REAL ; 
	MesQW	 : REAL ; 
	CalSW	: REAL ; 
	
	CalEacdelWh	: REAL ; 
	CalEarecWh	: REAL ; 	
	CalEreacdelvah	: REAL ; 
	CalErearecvah	: REAL ; 

	
END_VAR
//INITIALIZING MODBUS REQUESTS //
	FB_ModbusRead_I1[1](Reset:= CmdClearFault_G ,sIPAddr:=ParamIpAddress, tTimeout:= ParamTimeout,nTcpPort:=502);

// CP-Read / Write 



IF MesDataExd.MesData.MesCP_Read  THEN	
// MODBUS REQUEST//
	FB_ModbusRead_I1[1](
		nQuantity		:= 122, 
		nMBAddr			:= 19000, 
		nUnitID			:= ParamUnitID,
		cbLength		:= SIZEOF(MesBlock1_Temp) , 
		pDestAddr		:= ADR(MesBlock1_Temp) ,
		ClockRead		:= MesDataExd.MesData.MesCP_Read AND ClockRead ,
		ModbusReadAlarm	=>	MesModbusReadAlarm[1] , 
		ErrorId			=> MesModbusAlarmCode);

// PROPERTIES UPDATE // 


	// Block 1
MW( WORD_STRONG:= MesBlock1_Temp[26], WORD_WEAK := MesBlock1_Temp[27], VAR_OUT:=MesPW);
MW( WORD_STRONG:= MesBlock1_Temp[42], WORD_WEAK := MesBlock1_Temp[43], VAR_OUT:=MesQW);
MW( WORD_STRONG:= MesBlock1_Temp[44], WORD_WEAK := MesBlock1_Temp[45], VAR_OUT:=MesDataExd.MesData.MesCosPhi1);
MW( WORD_STRONG:= MesBlock1_Temp[46], WORD_WEAK := MesBlock1_Temp[47], VAR_OUT:=MesDataExd.MesData.MesCosPhi2);
MW( WORD_STRONG:= MesBlock1_Temp[48], WORD_WEAK := MesBlock1_Temp[49], VAR_OUT:=MesDataExd.MesData.MesCosPhi3);
MW( WORD_STRONG:= MesBlock1_Temp[0], WORD_WEAK := MesBlock1_Temp[1], VAR_OUT:=MesDataExd.MesData.MesV1);
MW( WORD_STRONG:= MesBlock1_Temp[2], WORD_WEAK := MesBlock1_Temp[3], VAR_OUT:=MesDataExd.MesData.MesV2);
MW( WORD_STRONG:= MesBlock1_Temp[4], WORD_WEAK := MesBlock1_Temp[5], VAR_OUT:=MesDataExd.MesData.MesV3);
MW( WORD_STRONG:= MesBlock1_Temp[6], WORD_WEAK := MesBlock1_Temp[7], VAR_OUT:=MesDataExd.MesData.MesU12);
MW( WORD_STRONG:= MesBlock1_Temp[8], WORD_WEAK := MesBlock1_Temp[9], VAR_OUT:=MesDataExd.MesData.MesU23);
MW( WORD_STRONG:= MesBlock1_Temp[10], WORD_WEAK := MesBlock1_Temp[11], VAR_OUT:=MesDataExd.MesData.MesU31);
MW( WORD_STRONG:= MesBlock1_Temp[12], WORD_WEAK := MesBlock1_Temp[13], VAR_OUT:=MesDataExd.MesData.MesI1);
MW( WORD_STRONG:= MesBlock1_Temp[14], WORD_WEAK := MesBlock1_Temp[15], VAR_OUT:=MesDataExd.MesData.MesI2);
MW( WORD_STRONG:= MesBlock1_Temp[16], WORD_WEAK := MesBlock1_Temp[17], VAR_OUT:=MesDataExd.MesData.MesI3);
MW( WORD_STRONG:= MesBlock1_Temp[50], WORD_WEAK := MesBlock1_Temp[51], VAR_OUT:=MesDataExd.MesData.MesFreq);

MW( WORD_STRONG:= MesBlock1_Temp[20], WORD_WEAK := MesBlock1_Temp[21], VAR_OUT:=MesP1W);
MW( WORD_STRONG:= MesBlock1_Temp[22], WORD_WEAK := MesBlock1_Temp[23], VAR_OUT:=MesP2W);
MW( WORD_STRONG:= MesBlock1_Temp[24], WORD_WEAK := MesBlock1_Temp[25], VAR_OUT:=MesP3W);
MW( WORD_STRONG:= MesBlock1_Temp[36], WORD_WEAK := MesBlock1_Temp[37], VAR_OUT:=MesQ1W);
MW( WORD_STRONG:= MesBlock1_Temp[38], WORD_WEAK := MesBlock1_Temp[39], VAR_OUT:=MesQ2W);
MW( WORD_STRONG:= MesBlock1_Temp[40], WORD_WEAK := MesBlock1_Temp[41], VAR_OUT:=MesQ3W);
MW( WORD_STRONG:= MesBlock1_Temp[34], WORD_WEAK := MesBlock1_Temp[35], VAR_OUT:=CalSW);


MW( WORD_STRONG:= MesBlock1_Temp[68], WORD_WEAK := MesBlock1_Temp[69], VAR_OUT:=CalEarecWh);
MW( WORD_STRONG:= MesBlock1_Temp[76], WORD_WEAK := MesBlock1_Temp[74], VAR_OUT:=CalEacdelWh);
MW( WORD_STRONG:= MesBlock1_Temp[100], WORD_WEAK := MesBlock1_Temp[101], VAR_OUT:=CalErearecvah);
MW( WORD_STRONG:= MesBlock1_Temp[108], WORD_WEAK := MesBlock1_Temp[109], VAR_OUT:=CalEreacdelvah);




// Properties Update 	
MesDataExd.MesData.MesP		:= MesPW / 1000 ; // kW 
MesDataExd.MesData.MesP1		:= MesP1W / 1000 ; 
MesDataExd.MesData.MesP2       := MesP2W / 1000 ; 
MesDataExd.MesData.MesP3       := MesP3W / 1000 ; 
MesDataExd.MesData.MesQ        := MesQW / 1000 ; 
MesDataExd.MesData.MesQ1       := MesQ1W / 1000 ; 
MesDataExd.MesData.MesQ2       := MesQ2W / 1000 ; 
MesDataExd.MesData.MesQ3       := MesQ3W / 1000 ; 
MesDataExd.MesData.MesS		:= CalSW / 1000 ; 

MesDataExd.MesData.MesEActProd		:= CalEacdelWh /1000 ; // kWh 
MesDataExd.MesData.MesEActCons		:= CalEarecWh / 1000 ; 
MesDataExd.MesData.MesEReactProd	:= CalEreacdelvah /1000 ; 
MesDataExd.MesData.MesEReactCons	:= CalErearecvah / 1000  ; 
END_IF 

MesDataExd.MesData.MesCosPhi    := (MesDataExd.MesData.MesCosPhi1 + MesDataExd.MesData.MesCosPhi2 + MesDataExd.MesData.MesCosPhi3)/3;
MesDataExd.MesData.MesI 		:= (MesDataExd.MesData.MesI1 + MesDataExd.MesData.MesI2 + MesDataExd.MesData.MesI3 )/3 ; 
MesDataExd.MesData.MesU			:= (MesDataExd.MesData.MesU12 + MesDataExd.MesData.MesU23 + MesDataExd.MesData.MesU31 ) /3 ; 
MesDataExd.MesData.MesV			:= (MesDataExd.MesData.MesV1 + MesDataExd.MesData.MesV2 + MesDataExd.MesData.MesV3 ) /3 ;

MesDataExd.MesData.MesCosPhi     := (MesDataExd.MesData.MesCosPhi1 + MesDataExd.MesData.MesCosPhi2 + MesDataExd.MesData.MesCosPhi3)/3;
MesDataExd.MesData.MesI :=  ( MesDataExd.MesData.MesI1 + MesDataExd.MesData.MesI2 + MesDataExd.MesData.MesI3 )/3 ; 
MesDataExd.MesData.MesU		:= 	(MesDataExd.MesData.MesU12 + MesDataExd.MesData.MesU23 + MesDataExd.MesData.MesU31 ) /3 ; 
MesDataExd.MesData.MesV		:= 	(MesDataExd.MesData.MesV1 + MesDataExd.MesData.MesV2 + MesDataExd.MesData.MesV3 ) /3 ; 

IF MesDataExd.MesData.MesP > 0.01 OR MesDataExd.MesData.MesP < -0.01 THEN
MesDataExd.MesData.MesTanPhi := MesDataExd.MesData.MesQ /MesDataExd.MesData.MesP;
ELSE
MesDataExd.MesData.MesTanPhi := 0;
END_IF
END_METHOD

END_FUNCTION_BLOCK

// ---- 01_Equipement_Library/Operation Meter/FB_PM_PM800.TcPOU
FUNCTION_BLOCK FB_PM_PM800 EXTENDS FB_PM_Base
VAR_INPUT PERSISTENT
	{attribute 'OPC.UA.DA' := '1'} 
	ParamIPAddress 	: STRING;	(* (NA) IP Adress of PM 800.*)
	
END_VAR

VAR_INPUT
	MesDataExd AT %Q*	: PM_PM800 ;
END_VAR

VAR_OUTPUT
END_VAR
VAR

	
	// Modbus Read Variables
	FB_ModbusReadAI : ARRAY[1..2] OF FB_ModbusRead ;
	
	// Temp Blocks Filled by Requests
	AI_List_1 	    : ARRAY[1..128] OF WORD ;
	AI_List_2 		: ARRAY[1..128] OF WORD ;
	
	tTimeout 		: TIME := T#2S ;
	
END_VAR

METHOD M_AlarmManagement
VAR_INPUT
END_VAR
//////////////////
// Digiware measurement tool alarm and warning management
/////////////////

VAR 
	// Method local variables (reinitialized at each cycle) 
	FB_AlarmCodeManager			: FB_AlarmCodeManager ; 
	
	ComWarning					: BOOL;			// Error in one of the Modbus Requests
	ComAlarm					: BOOL;			// Error in both Modbus Requests
	
END_VAR
ComWarning 	:= FB_ModbusReadAI[1].ModbusReadAlarm OR FB_ModbusReadAI[2].ModbusReadAlarm;
ComAlarm 	:= FB_ModbusReadAI[1].ModbusReadAlarm AND FB_ModbusReadAI[2].ModbusReadAlarm;
	
TON_ComAlarm(IN:= ComAlarm , PT:= ParamTempoComAlarm, Q=> MesDataExd.MesData.MesAlarmCom) ;	
TON_ComWarning(IN:= ComWarning  , PT:= ParamTempoComAlarm, Q=>MesWarningCom) ;	

//					General com alarm : All the read FB fucked up


// ALARM CODE //
	FB_AlarmCodeManager(
		bAlarm1			:= MesDataExd.MesData.MesAlarmCom  , 					// Communication Alarm #COM
		bAlarm2			:=FALSE, // 
		bAlarm3			:=FALSE, // 
		bAlarm4			:=FALSE, // 
		bAlarm5			:=FALSE, //
		bAlarm6			:=FALSE, //
		bAlarm7			:=FALSE, //
		bAlarm8			:=FALSE, //
		bAlarm9			:=FALSE, //
		bAlarm10		:=FALSE, //
		bAlarm11		:=FALSE, //
		bAlarm12		:=FALSE, //
		bAlarm13		:=FALSE, //
		bAlarm14		:=FALSE, //
		bAlarm15		:= FALSE , 			// 			 
		wAlarmCode		=>MesDataExd.MesData.MesAlarmCode);

// WARNING CODE //
	FB_AlarmCodeManager(		
		bAlarm1			:=MesWarningCom	,				 // Communication Warning #COM
		bAlarm2			:=FALSE, 		// 
		bAlarm3			:=FALSE, 		// 
		bAlarm4			:=FALSE, 		// 
		bAlarm5			:=FALSE, //
		bAlarm6			:=FALSE, //
		bAlarm7			:=FALSE, //
		bAlarm8			:=FALSE, //
		bAlarm9			:=FALSE, //
		bAlarm10		:=FALSE, //
		bAlarm11		:=FALSE, //
		bAlarm12		:=FALSE, //
		bAlarm13		:=FALSE, //
		bAlarm14		:=FALSE, //
		bAlarm15		:=FALSE, //
		wAlarmCode		=>MesDataExd.MesData.MesWarningCode);		

// EVENT CODE //
END_METHOD

METHOD M_CP
//////////////////
//  Emulator
/////////////////

VAR 
	// Method local variables (reinitialized at each cycle) 
	
END_VAR


SUPER^.M_CP() ; 




Trig_Cmd_Read(CLK:=IN_CmdToggleRead);
	
IF Trig_Cmd_Read.Q THEN
	IN_CmdToggleRead := FALSE;
	MesDataExd.MesData.MesCP_Read := NOT MesDataExd.MesData.MesCP_Read;
END_IF
END_METHOD

METHOD M_Read
VAR_INPUT
END_VAR
VAR
	MW					: FB_MergeWordsToDint;
	Test : REAL;
END_VAR
// CP-Read / Write 



IF MesDataExd.MesData.MesCP_Read  THEN	

// Analogic Inputs Modbus Requests
	
	FB_ModbusReadAI[1](pDestAddr := ADR(AI_List_1),
					sIPAddr := ParamIPAddress,
					tTimeout := tTimeout,
					nTcpPort := 502,
					nQuantity := 110,
					nMBAddr := 1099,
					cbLength := SIZEOF(AI_List_1),
					nUnitID := 1,
					ClockRead := MesDataExd.MesData.MesCP_Read AND ClockRead,
					Reset := CmdClearFault_G OR IN_CmdReset_L);
					
	FB_ModbusReadAI[2](pDestAddr := ADR(AI_List_2),
					sIPAddr := ParamIPAddress,
					tTimeout := tTimeout,
					nTcpPort := 502,
					nQuantity := 18,
					nMBAddr := 1699,
					cbLength := SIZEOF(AI_List_2),
					nUnitID := 1,
					ClockRead := MesDataExd.MesData.MesCP_Read AND ClockRead,
					Reset := CmdClearFault_G OR IN_CmdReset_L);
				
	//  MesDataExd.MesData.Filling Analogic Data			           
													
	MW(WORD_STRONG :=  AI_List_1[1  ],	WORD_WEAK := AI_List_1[1  ], SIZE := 1, FIX := 0, SIGNED := 0, VAR_OUT	:= MesDataExd.MesData.MesI1);
	MW(WORD_STRONG :=  AI_List_1[2  ],	WORD_WEAK := AI_List_1[2  ], SIZE := 1, FIX := 0, SIGNED := 0, VAR_OUT	:= MesDataExd.MesData.MesI2);
	MW(WORD_STRONG :=  AI_List_1[3  ],	WORD_WEAK := AI_List_1[3  ], SIZE := 1, FIX := 0, SIGNED := 0, VAR_OUT	:= MesDataExd.MesData.MesI3);
	MW(WORD_STRONG :=  AI_List_1[6  ],	WORD_WEAK := AI_List_1[6  ], SIZE := 1, FIX := 0, SIGNED := 0, VAR_OUT	:= MesDataExd.MesData.MesI);
	MW(WORD_STRONG :=  AI_List_1[21 ],	WORD_WEAK := AI_List_1[21 ], SIZE := 1, FIX := 0, SIGNED := 0, VAR_OUT	:= MesDataExd.MesData.MesU12);
	MW(WORD_STRONG :=  AI_List_1[22 ],	WORD_WEAK := AI_List_1[22 ], SIZE := 1, FIX := 0, SIGNED := 0, VAR_OUT	:= MesDataExd.MesData.MesU23);
	MW(WORD_STRONG :=  AI_List_1[23 ],	WORD_WEAK := AI_List_1[23 ], SIZE := 1, FIX := 0, SIGNED := 0, VAR_OUT	:= MesDataExd.MesData.MesU31);
	MW(WORD_STRONG :=  AI_List_1[44 ],	WORD_WEAK := AI_List_1[44 ], SIZE := 1, FIX := 0, SIGNED := 0, VAR_OUT	:= MesDataExd.MesData.MesP);
	MW(WORD_STRONG :=  AI_List_1[48 ],	WORD_WEAK := AI_List_1[48 ], SIZE := 1, FIX := 0, SIGNED := 0, VAR_OUT	:= MesDataExd.MesData.MesQ);
	MW(WORD_STRONG :=  AI_List_1[64 ],	WORD_WEAK := AI_List_1[64 ], SIZE := 1, FIX := 3, SIGNED := 0, VAR_OUT	:= MesDataExd.MesData.MesCosPhi);
	MW(WORD_STRONG :=  AI_List_1[81 ],	WORD_WEAK := AI_List_1[81 ], SIZE := 1, FIX := 0, SIGNED := 0, VAR_OUT	:= MesDataExd.MesData.MesFreq);
	
	MW(WORD_STRONG :=  AI_List_1[101],	WORD_WEAK := AI_List_1[101], SIZE := 1, FIX := 0, SIGNED := 0, VAR_OUT	:= MesDataExd.MesTHD1);
	MW(WORD_STRONG :=  AI_List_1[102],	WORD_WEAK := AI_List_1[102], SIZE := 1, FIX := 0, SIGNED := 0, VAR_OUT	:= MesDataExd.MesTHD2);
	MW(WORD_STRONG :=  AI_List_1[103],	WORD_WEAK := AI_List_1[103], SIZE := 1, FIX := 0, SIGNED := 0, VAR_OUT	:= MesDataExd.MesTHD3);
	MW(WORD_STRONG :=  AI_List_1[108],	WORD_WEAK := AI_List_1[108], SIZE := 1, FIX := 0, SIGNED := 0, VAR_OUT	:= MesDataExd.MesTHD1N);
	MW(WORD_STRONG :=  AI_List_1[109],	WORD_WEAK := AI_List_1[109], SIZE := 1, FIX := 0, SIGNED := 0, VAR_OUT	:= MesDataExd.MesTHD2N);
	MW(WORD_STRONG :=  AI_List_1[110],	WORD_WEAK := AI_List_1[110], SIZE := 1, FIX := 0, SIGNED := 0, VAR_OUT	:= MesDataExd.MesTHD3N);
	
	MesDataExd.MesData.MesEActProd 	:= (WORD_TO_REAL(AI_List_2[1  ]) + WORD_TO_REAL(AI_List_2[2  ])*10000 + WORD_TO_REAL(AI_List_2[3  ])*100000000 + WORD_TO_REAL(AI_List_2[4  ])*1000000000000)/1000;
	MesDataExd.MesData.MesEReactProd := (WORD_TO_REAL(AI_List_2[5  ]) + WORD_TO_REAL(AI_List_2[6  ])*10000 + WORD_TO_REAL(AI_List_2[7  ])*100000000 + WORD_TO_REAL(AI_List_2[8  ])*1000000000000)/1000;
	MesDataExd.MesData.MesEActCons 	:= (WORD_TO_REAL(AI_List_2[9  ]) + WORD_TO_REAL(AI_List_2[10 ])*10000 + WORD_TO_REAL(AI_List_2[11 ])*100000000 + WORD_TO_REAL(AI_List_2[12  ])*1000000000000)/1000;
	MesDataExd.MesData.MesEReactCons := (WORD_TO_REAL(AI_List_2[13 ]) + WORD_TO_REAL(AI_List_2[14 ])*10000 + WORD_TO_REAL(AI_List_2[15 ])*100000000 + WORD_TO_REAL(AI_List_2[16  ])*1000000000000)/1000;	


END_IF
END_METHOD

END_FUNCTION_BLOCK

// ---- 01_Equipement_Library/Operation Meter/FB_PM_Q100.TcPOU
FUNCTION_BLOCK FB_PM_Q100 EXTENDS FB_PM_Base
VAR_INPUT PERSISTENT
		ParamIPAddress				: STRING 	:= '192.168.20.66'; 	(* (NA)Config: IP Adress of PV INverter	*)
		ParamUnitID 				: BYTE  	:= 1; 			  		(* (NA)   Modbus Unit ID.               *)
		ParamTCPPort				: UINT		:= 502;					(* (NA) TCP port for modbus             *)

END_VAR

VAR_INPUT 
		MesDataExd			: PM_Q100;
END_VAR

VAR_OUTPUT
END_VAR
VAR
	// M_READ VARIABLES//

		AX_SB						: ARRAY [1..CstNbSB_INV_G] OF JuncBox;
		AX_ModbusRead		   		: ARRAY [1..3] OF FB_ModbusRead ; 					// (NA) FB for Modbus Reading
		
		MesBlock1_Temp 				: ARRAY[1..2]  OF WORD; 			// (NA) Temporary Block with multiple modbus reading (Caution : Double Word variables)
		MesBlock2_Temp 				: ARRAY[1..76]  OF WORD; 			// (NA) Temporary Block with multiple modbus reading (Caution : Double Word variables)
		MesBlock3_Temp 				: ARRAY[1..38]  OF WORD; 			// (NA) Temporary Block with multiple modbus reading (Caution : Double Word variables)

		AX_ReadAlarm 		  		: ARRAY [1..3] OF BOOL ; 							// (NA) Modbus Read Alarm for all modbus frames		
		AX_ReadAlarmCode			: ARRAY [1..3] OF UDINT;							// (NA) Modbus Read Alarm Code		
		AX_ReadBusy					: ARRAY [1..3] OF BOOL;								// (NA) Modbus Read Busy  
		AX_ReadCompleted			: ARRAY [1..3] OF BOOL;								// (NA) Modbus Read Completed
				
	

END_VAR

METHOD M_AlarmManagement
//////////////////
// Manages IntelliGen Alarms
/////////////////

VAR 
	// Method local variables (reinitialized at each cycle) 
	FB_AlarmCodeManager : FB_AlarmCodeManager ; 

	KK					: BYTE;		// For Loop 
	
	ComWarning			: BOOL;		// Aggregated Wcommunication warning
	ComAlarm			: BOOL;		// Aggregated communication Alarm

END_VAR
	//Alarm
	TON_ComAlarm(IN:= (AX_ModbusRead[1].ModbusReadAlarm) AND (AX_ModbusRead[2].ModbusReadAlarm) AND (AX_ModbusRead[3].ModbusReadAlarm) , PT:= ParamTempoComAlarm, Q=> MesDataExd.MesData.MesAlarmCom) ;	

	// Alarms if ALL MODBUS frames didn't work and timeout of 15s
	
	
// ALARM CODE //
	FB_AlarmCodeManager(
		bAlarm1			:= MesDataExd.MesData.MesAlarmCom,			// Communication general alarm (desactivate if LOC) 
		bAlarm2			:= FALSE,						//
		bAlarm3			:= FALSE, 						//
		bAlarm4			:= FALSE, 		            	//  
		bAlarm5			:= FALSE, 						//
		bAlarm6			:= FALSE, 						//
		bAlarm7			:= False, 						//
		bAlarm8			:= False, 						//
		bAlarm9			:= FALSE, 						//
		bAlarm10		:= FALSE, 						//
		bAlarm11		:= FALSE,                       //
		bAlarm12		:= FALSE,                       //
		bAlarm13		:= FALSE,                       //
		bAlarm14		:= FALSE, 						//
		bAlarm15		:= FALSE, 		                //
		wAlarmCode		=>MesDataExd.MesData.MesAlarmCode);
END_METHOD

METHOD M_CP
//////////////////
//  Emulator
/////////////////

VAR 
	// Method local variables (reinitialized at each cycle) 
	
END_VAR


SUPER^.M_CP() ; 




Trig_Cmd_Read(CLK:=IN_CmdToggleRead);
	
IF Trig_Cmd_Read.Q THEN
	IN_CmdToggleRead := FALSE;
	MesDataExd.MesData.MesCP_Read := NOT MesDataExd.MesData.MesCP_Read;
END_IF
END_METHOD

METHOD M_Execute
//////////////////
//  Method Calls 
/////////////////

VAR 
	// Method local variables (reinitialized at each cycle) 

END_VAR
IF NOT bInit THEN
	M_Init();
END_IF


SUPER^.M_Execute() ;
END_METHOD

METHOD M_Read
//////////////////
//  Read Modbus Variable for PCS . 
/////////////////
VAR 
	// Method local variables (reinitialized at each cycle) 
		MW 					: FB_MergeWordsToFloat; 
		MW1					: FB_MergeWordsToDint;
		
	KK: INT;
	MesWarningCodeAkuo: INT;
	MesPTemp: REAL;
	MesQTemp: REAL;
END_VAR
// CP-Read / Write 

 

IF MesDataExd.MesData.MesCP_Read  THEN		
	
	AX_ModbusRead[1]
	(
		pDestAddr := ADR(MesBlock1_Temp),
		sIPAddr := ParamIPAddress,
		tTimeout := ParamTimeout,
		nQuantity := 2,
		ntcpport := ParamTCPPort,
		nMBAddr := 100,
		nUnitID := ParamUnitID,
		cbLength := SIZEOF(MesBlock1_Temp),
		ClockRead := ClockRead,
		Reset := CmdClearFault_G OR IN_CmdReset_L,
		ErrorId => AX_ReadAlarmCode[1],
		ModbusReadAlarm => AX_ReadAlarm[1],
		Busy => AX_ReadBusy[1]	
	);
	
	AX_ModbusRead[2]
	(
		pDestAddr := ADR(MesBlock2_Temp),
		sIPAddr := ParamIPAddress,
		tTimeout := ParamTimeout,
		nQuantity := 76,
		ntcpport := ParamTCPPort,
		nMBAddr := 200,
		nUnitID := ParamUnitID,
		cbLength := SIZEOF(MesBlock2_Temp),
		ClockRead := ClockRead,
		Reset := CmdClearFault_G OR IN_CmdReset_L,
		ErrorId => AX_ReadAlarmCode[2],
		ModbusReadAlarm => AX_ReadAlarm[2],
		Busy => AX_ReadBusy[2]	
	);
	
	AX_ModbusRead[3]
	(
		pDestAddr := ADR(MesBlock3_Temp),
		sIPAddr := ParamIPAddress,
		tTimeout := ParamTimeout,
		nQuantity := 38,
		ntcpport := ParamTCPPort,
		nMBAddr := 800,
		nUnitID := ParamUnitID,
		cbLength := SIZEOF(MesBlock3_Temp),
		ClockRead := ClockRead,
		Reset := CmdClearFault_G OR IN_CmdReset_L,
		ErrorId => AX_ReadAlarmCode[3],
		ModbusReadAlarm => AX_ReadAlarm[3],
		Busy => AX_ReadBusy[3]	
	);
	
	FOR KK := 1 TO 3 DO
		AX_ReadCompleted[KK] := NOT AX_ReadAlarm[KK] AND NOT AX_ReadBusy[KK];
	END_FOR
	
MesDataExd.MesState1 := MesBlock1_Temp[1];
MesDataExd.MesState2 := MesBlock1_Temp[2];
	
	MW( WORD_STRONG:= MesBlock2_Temp[ 1], 	WORD_WEAK := MesBlock2_Temp[ 2],	VAR_OUT := MesDataExd.MesData.MesV1);
	MW( WORD_STRONG:= MesBlock2_Temp[ 3], 	WORD_WEAK := MesBlock2_Temp[ 4],	VAR_OUT := MesDataExd.MesData.MesV2);
	MW( WORD_STRONG:= MesBlock2_Temp[ 5], 	WORD_WEAK := MesBlock2_Temp[ 6],	VAR_OUT := MesDataExd.MesData.MesV3);
	MW( WORD_STRONG:= MesBlock2_Temp[ 7], 	WORD_WEAK := MesBlock2_Temp[ 8],	VAR_OUT := MesDataExd.MesVN);
	MW( WORD_STRONG:= MesBlock2_Temp[ 9], 	WORD_WEAK := MesBlock2_Temp[10],	VAR_OUT := MesDataExd.MesData.MesI1);
	MW( WORD_STRONG:= MesBlock2_Temp[11], 	WORD_WEAK := MesBlock2_Temp[12],	VAR_OUT := MesDataExd.MesData.MesI2);
	MW( WORD_STRONG:= MesBlock2_Temp[13], 	WORD_WEAK := MesBlock2_Temp[14],	VAR_OUT := MesDataExd.MesData.MesI3);
	MW( WORD_STRONG:= MesBlock2_Temp[15], 	WORD_WEAK := MesBlock2_Temp[16],	VAR_OUT := MesDataExd.MesData.MesIN);
	MW( WORD_STRONG:= MesBlock2_Temp[17], 	WORD_WEAK := MesBlock2_Temp[18], 	VAR_OUT := MesDataExd.MesData.MesU12);
	MW( WORD_STRONG:= MesBlock2_Temp[19], 	WORD_WEAK := MesBlock2_Temp[20], 	VAR_OUT := MesDataExd.MesData.MesU23);
	MW( WORD_STRONG:= MesBlock2_Temp[21], 	WORD_WEAK := MesBlock2_Temp[22], 	VAR_OUT := MesDataExd.MesData.MesU31);
	MW( WORD_STRONG:= MesBlock2_Temp[23], 	WORD_WEAK := MesBlock2_Temp[24],  VAR_OUT := MesDataExd.MesData.MesV);
	MW( WORD_STRONG:= MesBlock2_Temp[25], 	WORD_WEAK := MesBlock2_Temp[26],  VAR_OUT := MesDataExd.MesData.MesI);
	MW( WORD_STRONG:= MesBlock2_Temp[27], 	WORD_WEAK := MesBlock2_Temp[28],  VAR_OUT := MesDataExd.MesData.MesP1);
	MW( WORD_STRONG:= MesBlock2_Temp[29], 	WORD_WEAK := MesBlock2_Temp[30],  VAR_OUT := MesDataExd.MesData.MesP2);
	MW( WORD_STRONG:= MesBlock2_Temp[31], 	WORD_WEAK := MesBlock2_Temp[32],  VAR_OUT := MesDataExd.MesData.MesP3);
	MW( WORD_STRONG:= MesBlock2_Temp[33], 	WORD_WEAK := MesBlock2_Temp[34],  VAR_OUT := MesPTemp);
	MW( WORD_STRONG:= MesBlock2_Temp[35], 	WORD_WEAK := MesBlock2_Temp[36],  VAR_OUT := MesDataExd.MesData.MesQ1);
	MW( WORD_STRONG:= MesBlock2_Temp[37], 	WORD_WEAK := MesBlock2_Temp[38],  VAR_OUT := MesDataExd.MesData.MesQ2);
	MW( WORD_STRONG:= MesBlock2_Temp[39], 	WORD_WEAK := MesBlock2_Temp[40],  VAR_OUT := MesDataExd.MesData.MesQ3);
	MW( WORD_STRONG:= MesBlock2_Temp[41], 	WORD_WEAK := MesBlock2_Temp[42],  VAR_OUT := MesQTemp);
	MW( WORD_STRONG:= MesBlock2_Temp[43], 	WORD_WEAK := MesBlock2_Temp[44],  VAR_OUT := MesDataExd.MesData.MesS1);
	MW( WORD_STRONG:= MesBlock2_Temp[45], 	WORD_WEAK := MesBlock2_Temp[46],  VAR_OUT := MesDataExd.MesData.MesS2);
	MW( WORD_STRONG:= MesBlock2_Temp[47], 	WORD_WEAK := MesBlock2_Temp[48],  VAR_OUT := MesDataExd.MesData.MesS3);
	MW( WORD_STRONG:= MesBlock2_Temp[49], 	WORD_WEAK := MesBlock2_Temp[50],  VAR_OUT := MesDataExd.MesData.MesS);
	MW( WORD_STRONG:= MesBlock2_Temp[75], 	WORD_WEAK:= MesBlock2_Temp[76], VAR_OUT:= MesDataExd.MesData.MesFreq);
																			
																			
	MW( WORD_STRONG:= MesBlock3_Temp[01], 	WORD_WEAK := MesBlock3_Temp[02], VAR_OUT:= MesDataExd.MesEPerPulse);
	MW1( WORD_STRONG:= MesBlock3_Temp[07], 	WORD_WEAK := MesBlock3_Temp[08], Size := 2, fix := 0, signed := FALSE, VAR_OUT := MesDataExd.MesEac1_dmd);
	MW1( WORD_STRONG:= MesBlock3_Temp[09], 	WORD_WEAK := MesBlock3_Temp[10], Size := 2, fix := 0, signed := FALSE, VAR_OUT := MesDataExd.MesEac2_dmd);
	MW1( WORD_STRONG:= MesBlock3_Temp[11], 	WORD_WEAK := MesBlock3_Temp[12], Size := 2, fix := 0, signed := FALSE, VAR_OUT := MesDataExd.MesEac3_dmd);
	MW1( WORD_STRONG:= MesBlock3_Temp[13], 	WORD_WEAK := MesBlock3_Temp[14], Size := 2, fix := 0, signed := FALSE, VAR_OUT := MesDataExd.MesEac_dmd );
	MW1( WORD_STRONG:= MesBlock3_Temp[15], 	WORD_WEAK := MesBlock3_Temp[16], Size := 2, fix := 0, signed := FALSE, VAR_OUT := MesDataExd.MesEac1_sup);
	MW1( WORD_STRONG:= MesBlock3_Temp[17], 	WORD_WEAK := MesBlock3_Temp[18], Size := 2, fix := 0, signed := FALSE, VAR_OUT := MesDataExd.MesEac2_sup);
	MW1( WORD_STRONG:= MesBlock3_Temp[19], 	WORD_WEAK := MesBlock3_Temp[20], Size := 2, fix := 0, signed := FALSE, VAR_OUT := MesDataExd.MesEac3_sup);
	MW1( WORD_STRONG:= MesBlock3_Temp[21], 	WORD_WEAK := MesBlock3_Temp[22], Size := 2, fix := 0, signed := FALSE, VAR_OUT := MesDataExd.MesEac_sup );
	MW1( WORD_STRONG:= MesBlock3_Temp[23], 	WORD_WEAK := MesBlock3_Temp[24], Size := 2, fix := 0, signed := FALSE, VAR_OUT := MesDataExd.MesEreac1_ind);
	MW1( WORD_STRONG:= MesBlock3_Temp[25], 	WORD_WEAK := MesBlock3_Temp[26], Size := 2, fix := 0, signed := FALSE, VAR_OUT := MesDataExd.MesEreac2_ind);
	MW1( WORD_STRONG:= MesBlock3_Temp[27], 	WORD_WEAK := MesBlock3_Temp[28], Size := 2, fix := 0, signed := FALSE, VAR_OUT := MesDataExd.MesEreac3_ind);
	MW1( WORD_STRONG:= MesBlock3_Temp[29], 	WORD_WEAK := MesBlock3_Temp[30], Size := 2, fix := 0, signed := FALSE, VAR_OUT := MesDataExd.MesEreac_ind );
	MW1( WORD_STRONG:= MesBlock3_Temp[31], 	WORD_WEAK := MesBlock3_Temp[32], Size := 2, fix := 0, signed := FALSE, VAR_OUT := MesDataExd.MesEreac1_cap);
	MW1( WORD_STRONG:= MesBlock3_Temp[33], 	WORD_WEAK := MesBlock3_Temp[34], Size := 2, fix := 0, signed := FALSE, VAR_OUT := MesDataExd.MesEreac2_cap);
	MW1( WORD_STRONG:= MesBlock3_Temp[35], 	WORD_WEAK := MesBlock3_Temp[36], Size := 2, fix := 0, signed := FALSE, VAR_OUT := MesDataExd.MesEreac3_cap);
	MW1( WORD_STRONG:= MesBlock3_Temp[37], 	WORD_WEAK := MesBlock3_Temp[38], Size := 2, fix := 0, signed := FALSE, VAR_OUT := MesDataExd.MesEreac_cap);
	
MesDataExd.CalEac1_dmd      := MesDataExd.MesEac1_dmd        * MesDataExd.MesEPerPulse ;
MesDataExd.CalEac2_dmd      := MesDataExd.MesEac2_dmd        * MesDataExd.mesEperpulse ;
MesDataExd.CalEac3_dmd      := MesDataExd.MesEac3_dmd        * MesDataExd.mesEperpulse ;
MesDataExd.CalEac_dmd       := MesDataExd.MesEac_dmd         * MesDataExd.mesEperpulse ;
MesDataExd.CalEac1_sup      := MesDataExd.MesEac1_sup        * MesDataExd.mesEperpulse ;
MesDataExd.CalEac2_sup      := MesDataExd.MesEac2_sup        * MesDataExd.mesEperpulse ;
MesDataExd.CalEac3_sup      := MesDataExd.MesEac3_sup        * MesDataExd.mesEperpulse ;
MesDataExd.CalEac_sup       := MesDataExd.MesEac_sup         * MesDataExd.mesEperpulse ;
MesDataExd.CalEreac1_ind    := MesDataExd.MesEreac1_ind      * MesDataExd.mesEperpulse ;
MesDataExd.CalEreac2_ind    := MesDataExd.MesEreac2_ind      * MesDataExd.mesEperpulse ;
MesDataExd.CalEreac3_ind    := MesDataExd.MesEreac3_ind      * MesDataExd.mesEperpulse ;
MesDataExd.CalEreac_ind     := MesDataExd.MesEreac_ind       * MesDataExd.mesEperpulse ;
MesDataExd.CalEreac1_cap    := MesDataExd.MesEreac1_cap      * MesDataExd.mesEperpulse ;
MesDataExd.CalEreac2_cap    := MesDataExd.MesEreac2_cap      * MesDataExd.mesEperpulse ;
MesDataExd.CalEreac3_cap    := MesDataExd.MesEreac3_cap      * MesDataExd.mesEperpulse ;
MesDataExd.CalEreac_cap     := MesDataExd.MesEreac_cap       * MesDataExd.mesEperpulse ;
	
	// Changement signe P 
	
MesDataExd.MesData.MesP := -MesPTemp/1000;
MesDataExd.MesData.MesQ := -MesQTemp/1000;
MesDataExd.MesData.MesU := SQRT(3)*MesDataExd.MesData.MesV;
	
	IF ABS(MesDataExd.MesData.MesP) > 0 THEN
	MesDataExd.MesData.MesTanPhi := MesDataExd.MesData.MesQ / ABS(MesDataExd.MesData.MesP);
	END_IF


END_IF
END_METHOD

END_FUNCTION_BLOCK

// ---- 01_Equipement_Library/Operation Meter/FB_PM_SM103E.TcPOU
FUNCTION_BLOCK FB_PM_SM103E EXTENDS FB_PM_Base
//////////////////
// Measurement Solution based on Digiware, but access through PMS Socomec
//////////////////
VAR CONSTANT
	// Characteristics of the object (Same for all instances)
			
END_VAR

VAR_INPUT PERSISTENT
	// Parameters of the Object (instance specific) 
	{attribute 'OPC.UA.DA' := '1'} 
	ParamUnitID					: BYTE 		:= 5 ;								// (NA)unit ID
	

END_VAR

VAR_OUTPUT
	//Child objects
	
END_VAR

VAR_INPUT
		MesDataExd AT %Q*			: PM_Standard ;
END_VAR

VAR
	//M_ALARMMANAGEMENT VARIABLES//	                                                    							                                                								

	//M_READ VARIABLES//

	bReadError					: BOOL;
	bReadCompleted 				: BOOL;
	bReadBusy					: BOOL;
	InputStructRead 			: Struct_InputRTU;



	bReadError2					: BOOL;
	bReadCompleted2 				: BOOL;
	bReadBusy2					: BOOL;
	InputStructRead2 			: Struct_InputRTU;
	
	MesBlock1_Temp 				: ARRAY[1..64]  OF WORD; 		// (NA) Temporary Block with multiple mod
	MesBlock2_Temp 				: ARRAY[1..20]  OF WORD; 		// (NA) Temporary Block with multiple mod

		
		
	//M_INIT VARIABLES //
	
	// M_EXECUTE VARIABLES //
		RTrigI						: R_TRIG;



 
END_VAR

METHOD M_AlarmManagement
//////////////////
// Digiware measurement tool alarm and warning management
/////////////////

VAR 
	// Method local variables (reinitialized at each cycle) 
	FB_AlarmCodeManager			: FB_AlarmCodeManager ; 
	
	KK							: BYTE ;		// For loop
	
	CMWarning					: BOOL;			// At least one Digiware device in Alarm
	CMAlarm						: BOOL;			// At least one Digiware device in Alarm
	
END_VAR

CMAlarm := bReadError AND bReadError2 ; 
MesWarningCom := bReadError OR bReadError2 ;

//					General com alarm : All the read FB fucked up
TON_ComAlarm(IN:= CMAlarm , PT:= ParamTempoComAlarm, Q=>MesDataExd.MesData.MesAlarmCom) ;	 	// D50 LOC
// ALARM CODE //
	FB_AlarmCodeManager(
		bAlarm1			:= MesDataExd.MesData.MesAlarmCom   , 					// Communication Error  #COM
		bAlarm2			:=FALSE, 		// 
		bAlarm3			:=FALSE, 		// 
		bAlarm4			:=FALSE, 		// 
		bAlarm5			:=FALSE, 
		bAlarm6			:=FALSE, 
		bAlarm7			:=FALSE, 
		bAlarm8			:=FALSE, 
		bAlarm9			:=FALSE, 
		bAlarm10		:=FALSE, 
		bAlarm11		:=FALSE, 
		bAlarm12		:=FALSE, 
		bAlarm13		:=FALSE, 
		bAlarm14		:=FALSE, 
		bAlarm15		:= FALSE , 			// 							 
		wAlarmCode		=>MesDataExd.MesData.MesAlarmCode);

// WARNING CODE //
	FB_AlarmCodeManager(		
		bAlarm1			:=MesWarningCom	,				 // Communication warning #COM
		bAlarm2			:=FALSE, 		// 
		bAlarm3			:=FALSE, 		// 
		bAlarm4			:=FALSE, 		// 
		bAlarm5			:=FALSE, 
		bAlarm6			:=FALSE, 
		bAlarm7			:=FALSE, 
		bAlarm8			:=FALSE, 
		bAlarm9			:=FALSE, 
		bAlarm10		:=FALSE, 
		bAlarm11		:=FALSE, 
		bAlarm12		:=FALSE, 
		bAlarm13		:=FALSE, 
		bAlarm14		:=FALSE, 
		bAlarm15		:=FALSE, 
		wAlarmCode		=>MesDataExd.MesData.MesWarningCode);
END_METHOD

METHOD M_CP
//////////////////
//  Emulator
/////////////////

VAR 
	// Method local variables (reinitialized at each cycle) 
	
END_VAR


SUPER^.M_CP() ; 




Trig_Cmd_Read(CLK:=IN_CmdToggleRead);
	
IF Trig_Cmd_Read.Q THEN
	IN_CmdToggleRead := FALSE;
	MesDataExd.MesData.MesCP_Read := NOT MesDataExd.MesData.MesCP_Read;
END_IF
END_METHOD

METHOD M_Init
VAR 

END_VAR
END_METHOD

METHOD M_Read
//////////////////
//  Read Modbus Variable for PCS . 
/////////////////
VAR 
	// Method local variables (reinitialized at each cycle) 
	MW 					: FB_MergeWordsToDint; 
						// FOR Loop 


END_VAR
// CP-Read / Write 


IF MesDataExd.MesData.MesCP_Read  THEN	

(*
//Metrology

InputStructRead.InBuffer := ADR(MesBlock1_Temp);
InputStructRead.InFunction := 3;
InputStructRead.InQuantity := 54;
InputStructRead.InStartAddr := 768;
InputStructRead.InUnitID := ParamUnitID;

InputStructRead.OutBusy := ADR(bReadBusy);
InputStructRead.OutError := ADR(bReadError);
InputStructRead.OutCompleted := ADR(bReadCompleted);


RTrigI(CLK:= ClockRead );

IF RTrigI.Q THEN 
	A1_SUB_MV.ModbusRTU.M_AddAction_FIFO(InStruct:= InputStructRead , InPriority:=1 ) ; 
END_IF

// Properties update
MW(WORD_STRONG:=MesBlock1_Temp[1] , WORD_WEAK:=MesBlock1_Temp[2] , SIZE:=2, FIX :=3 , SIGNED :=FALSE , VAR_OUT := MesDataExd.MesData.MesI1  ); 
MW(WORD_STRONG:=MesBlock1_Temp[3] , WORD_WEAK:=MesBlock1_Temp[4] , SIZE:=2, FIX :=3 , SIGNED :=FALSE , VAR_OUT := MesDataExd.MesData.MesI2  ); 
MW(WORD_STRONG:=MesBlock1_Temp[5] , WORD_WEAK:=MesBlock1_Temp[6] , SIZE:=2, FIX :=3 , SIGNED :=FALSE , VAR_OUT := MesDataExd.MesData.MesI3  ); 
MW(WORD_STRONG:=MesBlock1_Temp[7] , WORD_WEAK:=MesBlock1_Temp[8] , SIZE:=2, FIX :=3 , SIGNED :=FALSE , VAR_OUT := MesDataExd.MesData.MesIN  ); 
MW(WORD_STRONG:=MesBlock1_Temp[9] , WORD_WEAK:=MesBlock1_Temp[10] , SIZE:=2, FIX :=2 , SIGNED :=FALSE , VAR_OUT := MesDataExd.MesData.MesU12  ); 
MW(WORD_STRONG:=MesBlock1_Temp[11] , WORD_WEAK:=MesBlock1_Temp[12] , SIZE:=2, FIX :=2 , SIGNED :=FALSE , VAR_OUT := MesDataExd.MesData.MesU23  ); 
MW(WORD_STRONG:=MesBlock1_Temp[13] , WORD_WEAK:=MesBlock1_Temp[14] , SIZE:=2, FIX :=2 , SIGNED :=FALSE , VAR_OUT := MesDataExd.MesData.MesU31  ); 
MW(WORD_STRONG:=MesBlock1_Temp[15] , WORD_WEAK:=MesBlock1_Temp[16] , SIZE:=2, FIX :=2 , SIGNED :=FALSE , VAR_OUT := MesDataExd.MesData.MesV1  ); 
MW(WORD_STRONG:=MesBlock1_Temp[17] , WORD_WEAK:=MesBlock1_Temp[18] , SIZE:=2, FIX :=2 , SIGNED :=FALSE , VAR_OUT := MesDataExd.MesData.MesV2  ); 
MW(WORD_STRONG:=MesBlock1_Temp[19] , WORD_WEAK:=MesBlock1_Temp[20] , SIZE:=2, FIX :=2 , SIGNED :=FALSE , VAR_OUT := MesDataExd.MesData.MesV3  ); 
MW(WORD_STRONG:=MesBlock1_Temp[21] , WORD_WEAK:=MesBlock1_Temp[22] , SIZE:=2, FIX :=2 , SIGNED :=FALSE , VAR_OUT := MesDataExd.MesData.MesFreq  ); 
MW(WORD_STRONG:=MesBlock1_Temp[23] , WORD_WEAK:=MesBlock1_Temp[24] , SIZE:=2, FIX :=2 , SIGNED :=TRUE , VAR_OUT := MesDataExd.MesData.MesP  ); 
MW(WORD_STRONG:=MesBlock1_Temp[25] , WORD_WEAK:=MesBlock1_Temp[26] , SIZE:=2, FIX :=2 , SIGNED :=TRUE , VAR_OUT := MesDataExd.MesData.MesQ  ); 
MW(WORD_STRONG:=MesBlock1_Temp[27] , WORD_WEAK:=MesBlock1_Temp[28] , SIZE:=2, FIX :=2 , SIGNED :=FALSE , VAR_OUT := MesDataExd.MesData.MesS  ); 
MW(WORD_STRONG:=MesBlock1_Temp[29] , WORD_WEAK:=MesBlock1_Temp[30] , SIZE:=2, FIX :=3 , SIGNED :=TRUE , VAR_OUT := MesDataExd.MesData.MesPF  ); 
MW(WORD_STRONG:=MesBlock1_Temp[31] , WORD_WEAK:=MesBlock1_Temp[32] , SIZE:=2, FIX :=2 , SIGNED :=TRUE , VAR_OUT := MesDataExd.MesData.MesP1  ); 
MW(WORD_STRONG:=MesBlock1_Temp[33] , WORD_WEAK:=MesBlock1_Temp[34] , SIZE:=2, FIX :=2 , SIGNED :=TRUE , VAR_OUT := MesDataExd.MesData.MesP2  ); 
MW(WORD_STRONG:=MesBlock1_Temp[35] , WORD_WEAK:=MesBlock1_Temp[36] , SIZE:=2, FIX :=2 , SIGNED :=TRUE , VAR_OUT := MesDataExd.MesData.MesP3  ); 
MW(WORD_STRONG:=MesBlock1_Temp[37] , WORD_WEAK:=MesBlock1_Temp[38] , SIZE:=2, FIX :=2 , SIGNED :=TRUE , VAR_OUT := MesDataExd.MesData.MesQ1  ); 
MW(WORD_STRONG:=MesBlock1_Temp[39] , WORD_WEAK:=MesBlock1_Temp[40] , SIZE:=2, FIX :=2 , SIGNED :=TRUE , VAR_OUT := MesDataExd.MesData.MesQ2  ); 
MW(WORD_STRONG:=MesBlock1_Temp[41] , WORD_WEAK:=MesBlock1_Temp[42] , SIZE:=2, FIX :=2 , SIGNED :=TRUE , VAR_OUT := MesDataExd.MesData.MesQ3  ); 
MW(WORD_STRONG:=MesBlock1_Temp[43] , WORD_WEAK:=MesBlock1_Temp[44] , SIZE:=2, FIX :=2 , SIGNED :=FALSE , VAR_OUT := MesDataExd.MesData.MesS1  ); 
MW(WORD_STRONG:=MesBlock1_Temp[45] , WORD_WEAK:=MesBlock1_Temp[46] , SIZE:=2, FIX :=2 , SIGNED :=FALSE , VAR_OUT := MesDataExd.MesData.MesS2  ); 
MW(WORD_STRONG:=MesBlock1_Temp[47] , WORD_WEAK:=MesBlock1_Temp[48] , SIZE:=2, FIX :=2 , SIGNED :=FALSE , VAR_OUT := MesDataExd.MesData.MesS3  ); 
MW(WORD_STRONG:=MesBlock1_Temp[49] , WORD_WEAK:=MesBlock1_Temp[50] , SIZE:=2, FIX :=3 , SIGNED :=TRUE , VAR_OUT := MesDataExd.MesData.MesPF1  ); 
MW(WORD_STRONG:=MesBlock1_Temp[51] , WORD_WEAK:=MesBlock1_Temp[52] , SIZE:=2, FIX :=3 , SIGNED :=TRUE , VAR_OUT := MesDataExd.MesData.MesPF2  ); 
MW(WORD_STRONG:=MesBlock1_Temp[53] , WORD_WEAK:=MesBlock1_Temp[54] , SIZE:=2, FIX :=3 , SIGNED :=TRUE , VAR_OUT := MesDataExd.MesData.MesPF3  ); 
 


MesData.MesI := MesDataExd.MesData.MesI1 + MesDataExd.MesData.MesI2 MesDataExd.MesData.MesI3 ) /3 ; 
MesData.MesU := MesDataExd.MesData.MesU12 + MesDataExd.MesData.MesU23 MesDataExd.MesData.MesU31 ) /3 ; 
MesData.MesV := MesDataExd.MesData.MesV1 + MesDataExd.MesData.MesV2 MesDataExd.MesData.MesV3 ) /3 ; 


//Energy
InputStructRead2.InBuffer := ADR(MesBlock2_Temp);
InputStructRead2.InFunction := 3;
InputStructRead2.InQuantity := 10;
InputStructRead2.InStartAddr := 50780;
InputStructRead2.InUnitID := ParamUnitID;

InputStructRead2.OutBusy := ADR(bReadBusy2);
InputStructRead2.OutError := ADR(bReadError2);
InputStructRead2.OutCompleted := ADR(bReadCompleted2);


IF RTrigI.Q THEN 
	A1_SUB_MV.ModbusRTU.M_AddAction_FIFO(InStruct:= InputStructRead2 , InPriority:=1 ) ; 
END_IF

// Properties update
MW(WORD_STRONG:=MesBlock2_Temp[1] , WORD_WEAK:=MesBlock2_Temp[2] , SIZE:=2, FIX :=0 , SIGNED :=FALSE , VAR_OUT := MesDataExd.MesData.MesEActProd  ); 
MW(WORD_STRONG:=MesBlock2_Temp[3] , WORD_WEAK:=MesBlock2_Temp[4] , SIZE:=2, FIX :=0 , SIGNED :=FALSE , VAR_OUT := MesDataExd.MesData.MesEReactProd  ); 

MW(WORD_STRONG:=MesBlock2_Temp[7] , WORD_WEAK:=MesBlock2_Temp[8] , SIZE:=2, FIX :=0 , SIGNED :=FALSE , VAR_OUT := MesDataExd.MesData.MesEActCons  ); 
MW(WORD_STRONG:=MesBlock2_Temp[9] , WORD_WEAK:=MesBlock2_Temp[10] , SIZE:=2, FIX :=0 , SIGNED :=FALSE , VAR_OUT := MesDataExd.MesData.MesEReactCons  ); 


*)

END_IF
END_METHOD

END_FUNCTION_BLOCK

// ---- 01_Equipement_Library/Operation Meter/FB_PM_PM3250.TcPOU
FUNCTION_BLOCK FB_PM_PM3250 EXTENDS FB_PM_Base
//////////////////
// Measurement Solution based on Digiware, but access through PMS Socomec
//////////////////
VAR CONSTANT
	// Characteristics of the object (Same for all instances)
			
END_VAR

VAR_INPUT PERSISTENT
	// Parameters of the Object (instance specific) 
	{attribute 'OPC.UA.DA' := '1'} 
	ParamUnitID					: BYTE 		:= 1 ;								(* (NA)unit ID*)
//	ParamInInterfaceSub			: BOOL := TRUE; 								// (NA) Serial interface RS422/RS485 TYPE (0:EL6021,1:SUB9)			
END_VAR

VAR_OUTPUT
	//Child objects
	
END_VAR

VAR_INPUT 
				MesDataExd AT %Q*				: PM_Standard ;
END_VAR

VAR

	//M_READ VARIABLES//
		InputStructRead 			: ARRAY[1..5] OF  Struct_InputRTU;

		AX_Quantity					: ARRAY[1..5] OF WORD;					// (NA) Quantity of blocks to read
		AX_Address					: ARRAY[1..5] OF WORD;					// (NA) Start address of the read
		MesBlock_Temp 				: ARRAY[1..5] OF ARRAY[1..125] OF WORD;	// (NA) Temporary Block with multiple modbus reading (U30 + I35)
		Busy						: BOOL;
		OutErrorMbRead				: ARRAY[1..5] OF BOOL;
	

	//M_INIT VARIABLES //
		OutFBCompleteted			: BOOL;
	// M_EXECUTE VARIABLES //
		RTrigI						: R_TRIG;

END_VAR

METHOD M_AlarmManagement
//////////////////
// Digiware measurement tool alarm and warning management
/////////////////

VAR 
	// Method local variables (reinitialized at each cycle) 
	FB_AlarmCodeManager			: FB_AlarmCodeManager ; 
	
	KK							: BYTE ;		// For loop
	
	CMWarning					: BOOL;			// At least one Digiware device in Alarm
	CMAlarm						: BOOL;			// At least one Digiware device in Alarm
	
END_VAR

	
TON_ComAlarm(IN:= OutErrorMbRead[1] AND OutErrorMbRead[2] AND OutErrorMbRead[3] AND OutErrorMbRead[4] AND OutErrorMbRead[5] , PT:= ParamTempoComAlarm, Q=> MesDataExd.MesData.MesAlarmCom) ;	
TON_ComWarning(IN:= OutErrorMbRead[1] OR OutErrorMbRead[2] OR OutErrorMbRead[3] OR OutErrorMbRead[4] OR OutErrorMbRead[5] , PT:= ParamTempoComAlarm, Q=>MesWarningCom) ;	

// General com alarm : All the read FB fucked up
// ALARM CODE //
	FB_AlarmCodeManager( 
		bAlarm1			:= MesDataExd.MesData.MesAlarmCom, 					// Communication Error  #COM
		bAlarm2			:=FALSE, 									// 
		bAlarm3			:=FALSE, 									// 
		bAlarm4			:=FALSE, 									// 
		bAlarm5			:=FALSE, 									//
		bAlarm6			:=FALSE, 									//
		bAlarm7			:=FALSE, 									//
		bAlarm8			:=FALSE, 									//
		bAlarm9			:=FALSE, 									//
		bAlarm10		:=FALSE, 									//
		bAlarm11		:=FALSE, 									//
		bAlarm12		:=FALSE, 									//
		bAlarm13		:=FALSE, 									//
		bAlarm14		:=FALSE, 									//
		bAlarm15		:= FALSE , 									//						 
		wAlarmCode		=>MesDataExd.MesData.MesAlarmCode);

// WARNING CODE //
	FB_AlarmCodeManager(		
		bAlarm1			:=	MesWarningCom,				 			// Communication Warning #COM	
		bAlarm2			:=FALSE, 									// 
		bAlarm3			:=FALSE, 									// 
		bAlarm4			:=FALSE, 									// 
		bAlarm5			:=FALSE, 									//
		bAlarm6			:=FALSE, 									//
		bAlarm7			:=FALSE, 									//
		bAlarm8			:=FALSE, 									//
		bAlarm9			:=FALSE, 									//
		bAlarm10		:=FALSE, 									//
		bAlarm11		:=FALSE, 									//
		bAlarm12		:=FALSE, 									//
		bAlarm13		:=FALSE, 									//
		bAlarm14		:=FALSE, 									//
		bAlarm15		:=FALSE, 									//
		wAlarmCode		=>MesDataExd.MesData.MesWarningCode);
END_METHOD

METHOD M_CP
//////////////////
//  Emulator
/////////////////

VAR 
	// Method local variables (reinitialized at each cycle) 
	
END_VAR


SUPER^.M_CP() ; 




Trig_Cmd_Read(CLK:=IN_CmdToggleRead);
	
IF Trig_Cmd_Read.Q THEN
	IN_CmdToggleRead := FALSE;
	MesDataExd.MesData.MesCP_Read := NOT MesDataExd.MesData.MesCP_Read;
END_IF
END_METHOD

METHOD M_Evaluate : BOOL
VAR_INPUT
END_VAR
END_METHOD

METHOD M_Execute
//////////////////
//  Method Calls 
/////////////////
VAR 
	// Method local variables (reinitialized at each cycle) 
	// EMULATOR
		Psoltot		: REAL;		// Total Solar Power . 
		KK			: BYTE;		// For Loop
	
END_VAR
// READING AND WRITING CLOCK //
	TP1(IN:=NOT TP1.Q , PT:= ParamClockReadTime);
	ClockRead 		:= TP1.Q;

// PERMANENT CONDITIONS //
	MesCP_Read 					:= TRUE  ; 
	
// METHODS CALLS //
	IF bInit THEN
		M_Init() ; 
		bInit							:= FALSE ; 
	ELSIF CmdInit_G OR IN_CmdReset_L THEN 
		bInit:= TRUE ;
	END_IF

	M_Read() ; 	
	M_AlarmManagement();
END_METHOD

METHOD M_Init
VAR 

END_VAR
	
AX_Quantity[1] := 12;
AX_Quantity[2] := 18;
AX_Quantity[3] := 32;
AX_Quantity[4] := 4;
AX_Quantity[5] := 32;

AX_Address[1]  := 2999;
AX_Address[2]  := 3020;
AX_Address[3]  := 3053;
AX_Address[4]  := 3107;
AX_Address[5]  := 3203;
END_METHOD

METHOD M_Read
//////////////////
//  Read Modbus Variable for PCS . 
/////////////////
VAR 
	// Method local variables (reinitialized at each cycle) 
	MW 					: FB_MergeWordsToFloat; 
	KK					: BYTE;  						// FOR Loop 
	MW2					: FB_MergeWordsToDint ; 

	
END_VAR
// CP-Read / Write 

 

IF MesDataExd.MesData.MesCP_Read  THEN	

	RTrigI(CLK:= ClockRead AND MesDataExd.MesData.MesCP_Read);
	//Metrology
	FOR KK:=1 TO 5 DO  
		InputStructRead[KK].InBuffer := ADR(MesBlock_Temp[KK]);
		InputStructRead[KK].InFunction := 3;
		InputStructRead[KK].InQuantity := AX_Quantity[KK];
		InputStructRead[KK].InStartAddr := AX_Address[KK];
		InputStructRead[KK].InUnitID := ParamUnitID;
		
		InputStructRead[KK].OutBusy := ADR(Busy);
		InputStructRead[KK].OutError := ADR(OutErrorMbRead[KK]);
		//InputStructRead[KK].OutCompleted := ADR(bReadCompleted);
		
		IF RTrigI.Q THEN 
			A1_SUBMV.FB_ModbusReadRTU.M_AddAction_FIFO(InStruct:= InputStructRead[KK] , InPriority:=1 ) ; 
		END_IF
		
	END_FOR 
	// PROPERTIES UPDATE // 
		// Block 1
	//MW( WORD_STRONG:= MesBlock_Temp[1][1], 	WORD_WEAK := MesBlock_Temp[1][2],	SIGNED:=TRUE, FIX:=0 , SIZE:=2, VAR_OUT := MesDataExd.MesData.MesI2);
		
	
	MW( WORD_STRONG:= MesBlock_Temp[1][1], 	WORD_WEAK := MesBlock_Temp[1][2], VAR_OUT := MesDataExd.MesData.MesI1);
	MW( WORD_STRONG:= MesBlock_Temp[1][3], 	WORD_WEAK := MesBlock_Temp[1][4], VAR_OUT:= MesDataExd.MesData.MesI2);
	MW( WORD_STRONG:= MesBlock_Temp[1][5], 	WORD_WEAK := MesBlock_Temp[1][6], VAR_OUT:= MesDataExd.MesData.MesI3);
	MW( WORD_STRONG:= MesBlock_Temp[1][7], 	WORD_WEAK := MesBlock_Temp[1][8], VAR_OUT:= MesDataExd.MesData.MesIN);
	MW( WORD_STRONG:= MesBlock_Temp[1][11], 	WORD_WEAK := MesBlock_Temp[1][12], VAR_OUT:= MesDataExd.MesData.MesI);
	
